LIN {X 0,Y 480.897,Z 537.281,A -85,B 0,C 180,E1 -6841.675,E2 -6841.675} C_VEL
LIN {X 0,Y 481.01,Z 535.652,A -85,B 0,C 180,E1 -6843.35,E2 -6843.35} C_VEL
LIN {X 0,Y 481.08,Z 532.877,A -85,B 0,C 180,E1 -6845.029,E2 -6845.029} C_VEL
LIN {X 0,Y 481.293,Z 528.594,A -85,B 0,C 180,E1 -6846.803,E2 -6846.803} C_VEL
LIN {X 0,Y 481.489,Z 523.502,A -85,B 0,C 180,E1 -6848.393,E2 -6848.393} C_VEL
LIN {X 0,Y 481.749,Z 516.626,A -85,B 0,C 180,E1 -6850.082,E2 -6850.082} C_VEL
LIN {X 0,Y 482.2,Z 509.189,A -85,B 0,C 180,E1 -6851.561,E2 -6851.561} C_VEL
LIN {X 0,Y 482.622,Z 500.167,A -85,B 0,C 180,E1 -6853.045,E2 -6853.045} C_VEL
LIN {X 0,Y 483.158,Z 490.915,A -85,B 0,C 180,E1 -6854.317,E2 -6854.317} C_VEL
LIN {X 0,Y 483.742,Z 479.844,A -85,B 0,C 180,E1 -6855.591,E2 -6855.591} C_VEL
LIN {X 0,Y 484.392,Z 467.732,A -85,B 0,C 180,E1 -6856.746,E2 -6856.746} C_VEL
LIN {X 0,Y 484.961,Z 455.431,A -85,B 0,C 180,E1 -6857.718,E2 -6857.718} C_VEL
LIN {X 0,Y 485.59,Z 440.986,A -85,B 0,C 180,E1 -6858.638,E2 -6858.638} C_VEL
LIN {X 0,Y 485.834,Z 427.276,A -85,B 0,C 180,E1 -6859.339,E2 -6859.339} C_VEL
LIN {X 0,Y 481.687,Z 414.112,A -85,B 0,C 180,E1 -6860.052,E2 -6860.052} C_VEL
LIN {X 0,Y 481.666,Z 414.111,A -85,B 0,C 180,E1 -6863.201,E2 -6863.201} C_VEL
LIN {X 0,Y 481.691,Z 414.114,A -85,B 0,C 180,E1 -6865.958,E2 -6865.958} C_VEL
LIN {X 0,Y 481.702,Z 414.107,A -85,B 0,C 180,E1 -6868.781,E2 -6868.781} C_VEL
LIN {X 0,Y 481.661,Z 414.113,A -85,B 0,C 180,E1 -6872.19,E2 -6872.19} C_VEL
LIN {X 0,Y 481.69,Z 414.107,A -85,B 0,C 180,E1 -6874.682,E2 -6874.682} C_VEL
LIN {X 0,Y 481.656,Z 414.115,A -85,B 0,C 180,E1 -6878.007,E2 -6878.007} C_VEL
LIN {X 0,Y 481.664,Z 414.113,A -85,B 0,C 180,E1 -6881.041,E2 -6881.041} C_VEL
LIN {X 0,Y 481.738,Z 414.259,A -85,B 0,C 180,E1 -6884.055,E2 -6884.055} C_VEL
LIN {X 0,Y 481.86,Z 418.445,A -85,B 0,C 180,E1 -6885.616,E2 -6885.616} C_VEL
LIN {X 0,Y 481.614,Z 430.552,A -85,B 0,C 180,E1 -6889.71,E2 -6889.71} C_VEL
LIN {X 0,Y 481.795,Z 440.07,A -85,B 0,C 180,E1 -6892.745,E2 -6892.745} C_VEL
LIN {X 0,Y 481.916,Z 449.965,A -85,B 0,C 180,E1 -6895.817,E2 -6895.817} C_VEL
LIN {X 0,Y 481.956,Z 459.783,A -85,B 0,C 180,E1 -6898.824,E2 -6898.824} C_VEL
LIN {X 0,Y 481.976,Z 469.257,A -85,B 0,C 180,E1 -6901.712,E2 -6901.712} C_VEL
LIN {X 0,Y 481.793,Z 479.207,A -85,B 0,C 180,E1 -6904.743,E2 -6904.743} C_VEL
LIN {X 0,Y 481.638,Z 488.806,A -85,B 0,C 180,E1 -6907.704,E2 -6907.704} C_VEL
LIN {X 0,Y 481.504,Z 497.467,A -85,B 0,C 180,E1 -6910.384,E2 -6910.384} C_VEL
LIN {X 0,Y 481.447,Z 502.384,A -85,B 0,C 180,E1 -6911.923,E2 -6911.923} C_VEL
LIN {X 0,Y 484.792,Z 518.216,A -85,B 0,C 180,E1 -6912.407,E2 -6912.407} C_VEL
LIN {X 0,Y 485.454,Z 522.705,A -85,B 0,C 180,E1 -6912.57,E2 -6912.57} C_VEL
LIN {X 0,Y 485.075,Z 535.599,A -85,B 0,C 180,E1 -6913.058,E2 -6913.058} C_VEL
LIN {X 0,Y 484.495,Z 549.866,A -85,B 0,C 180,E1 -6913.785,E2 -6913.785} C_VEL
LIN {X 0,Y 483.935,Z 562.713,A -85,B 0,C 180,E1 -6914.631,E2 -6914.631} C_VEL
LIN {X 0,Y 483.286,Z 574.358,A -85,B 0,C 180,E1 -6915.58,E2 -6915.58} C_VEL
LIN {X 0,Y 482.67,Z 585.939,A -85,B 0,C 180,E1 -6916.742,E2 -6916.742} C_VEL
LIN {X 0,Y 482.228,Z 596.661,A -85,B 0,C 180,E1 -6918.062,E2 -6918.062} C_VEL
LIN {X 0,Y 481.671,Z 606.186,A -85,B 0,C 180,E1 -6919.491,E2 -6919.491} C_VEL
LIN {X 0,Y 481.328,Z 614.151,A -85,B 0,C 180,E1 -6920.969,E2 -6920.969} C_VEL
LIN {X 0,Y 481.054,Z 620.547,A -85,B 0,C 180,E1 -6922.445,E2 -6922.445} C_VEL
LIN {X 0,Y 480.951,Z 626.202,A -85,B 0,C 180,E1 -6924.129,E2 -6924.129} C_VEL
LIN {X 0,Y 480.817,Z 630.31,A -85,B 0,C 180,E1 -6925.809,E2 -6925.809} C_VEL
LIN {X 0,Y 480.879,Z 631.825,A -85,B 0,C 180,E1 -6926.649,E2 -6926.649} C_VEL
LIN {X 0,Y 480.786,Z 633.83,A -85,B 0,C 180,E1 -6928.325,E2 -6928.325} C_VEL
LIN {X 0,Y 480.741,Z 634.5,A -85,B 0,C 180,E1 -6930,E2 -6930} C_VEL
LIN {X 0,Y 480.786,Z 633.827,A -85,B 0,C 180,E1 -6931.675,E2 -6931.675} C_VEL
LIN {X 0,Y 480.879,Z 631.826,A -85,B 0,C 180,E1 -6933.351,E2 -6933.351} C_VEL
LIN {X 0,Y 480.896,Z 628.445,A -85,B 0,C 180,E1 -6935.031,E2 -6935.031} C_VEL
LIN {X 0,Y 480.996,Z 623.596,A -85,B 0,C 180,E1 -6936.713,E2 -6936.713} C_VEL
LIN {X 0,Y 481.141,Z 618.859,A -85,B 0,C 180,E1 -6937.976,E2 -6937.976} C_VEL
LIN {X 0,Y 481.426,Z 612.055,A -85,B 0,C 180,E1 -6939.453,E2 -6939.453} C_VEL
LIN {X 0,Y 481.833,Z 603.569,A -85,B 0,C 180,E1 -6940.93,E2 -6940.93} C_VEL
LIN {X 0,Y 482.258,Z 593.829,A -85,B 0,C 180,E1 -6942.315,E2 -6942.315} C_VEL
LIN {X 0,Y 482.793,Z 583.991,A -85,B 0,C 180,E1 -6943.469,E2 -6943.469} C_VEL
LIN {X 0,Y 483.314,Z 573.157,A -85,B 0,C 180,E1 -6944.527,E2 -6944.527} C_VEL
LIN {X 0,Y 483.986,Z 561.269,A -85,B 0,C 180,E1 -6945.475,E2 -6945.475} C_VEL
LIN {X 0,Y 484.586,Z 548.033,A -85,B 0,C 180,E1 -6946.32,E2 -6946.32} C_VEL
LIN {X 0,Y 485.074,Z 535.108,A -85,B 0,C 180,E1 -6946.963,E2 -6946.963} C_VEL
LIN {X 0,Y 485.341,Z 521.153,A -85,B 0,C 180,E1 -6947.486,E2 -6947.486} C_VEL
LIN {X 0,Y 482.502,Z 507.123,A -85,B 0,C 180,E1 -6947.951,E2 -6947.951} C_VEL
LIN {X 0,Y 481.446,Z 502.32,A -85,B 0,C 180,E1 -6948.096,E2 -6948.096} C_VEL
LIN {X 0,Y 481.641,Z 492.574,A -85,B 0,C 180,E1 -6951.395,E2 -6951.395} C_VEL
LIN {X 0,Y 481.85,Z 483.299,A -85,B 0,C 180,E1 -6954.563,E2 -6954.563} C_VEL
LIN {X 0,Y 482.004,Z 475.751,A -85,B 0,C 180,E1 -6957.198,E2 -6957.198} C_VEL
LIN {X 0,Y 482.218,Z 468.781,A -85,B 0,C 180,E1 -6959.705,E2 -6959.705} C_VEL
LIN {X 0,Y 482.438,Z 460.823,A -85,B 0,C 180,E1 -6962.616,E2 -6962.616} C_VEL
LIN {X 0,Y 482.647,Z 452.865,A -85,B 0,C 180,E1 -6965.623,E2 -6965.623} C_VEL
LIN {X 0,Y 482.809,Z 444.905,A -85,B 0,C 180,E1 -6968.75,E2 -6968.75} C_VEL
LIN {X 0,Y 483.014,Z 438.229,A -85,B 0,C 180,E1 -6971.456,E2 -6971.456} C_VEL
LIN {X 0,Y 483.396,Z 429.907,A -85,B 0,C 180,E1 -6974.947,E2 -6974.947} C_VEL
LIN {X 0,Y 483.455,Z 425.426,A -85,B 0,C 180,E1 -6976.903,E2 -6976.903} C_VEL
LIN {X 0,Y 482.819,Z 420.482,A -85,B 0,C 180,E1 -6979.194,E2 -6979.194} C_VEL
LIN {X 0,Y 481.671,Z 414.114,A -85,B 0,C 180,E1 -6982.339,E2 -6982.339} C_VEL
LIN {X 0,Y 481.694,Z 414.11,A -85,B 0,C 180,E1 -6985.318,E2 -6985.318} C_VEL
LIN {X 0,Y 481.647,Z 414.118,A -85,B 0,C 180,E1 -6988.312,E2 -6988.312} C_VEL
LIN {X 0,Y 481.702,Z 414.111,A -85,B 0,C 180,E1 -6991.219,E2 -6991.219} C_VEL
LIN {X 0,Y 481.703,Z 414.101,A -85,B 0,C 180,E1 -6994.043,E2 -6994.043} C_VEL
LIN {X 0,Y 481.676,Z 414.11,A -85,B 0,C 180,E1 -6996.812,E2 -6996.812} C_VEL
LIN {X 0,Y 481.699,Z 414.1,A -85,B 0,C 180,E1 -6999.503,E2 -6999.503} C_VEL
LIN {X 0,Y 481.71,Z 414.108,A -85,B 0,C 180,E1 -7002.159,E2 -7002.159} C_VEL
LIN {X 0,Y 481.745,Z 414.097,A -85,B 0,C 180,E1 -7004.776,E2 -7004.776} C_VEL
LIN {X 0,Y 481.753,Z 414.102,A -85,B 0,C 180,E1 -7008.215,E2 -7008.215} C_VEL
LIN {X 0,Y 481.743,Z 414.095,A -85,B 0,C 180,E1 -7011.611,E2 -7011.611} C_VEL
LIN {X 0,Y 481.819,Z 414.095,A -85,B 0,C 180,E1 -7014.14,E2 -7014.14} C_VEL
LIN {X 0,Y 481.93,Z 414.073,A -85,B 0,C 180,E1 -7017.493,E2 -7017.493} C_VEL
LIN {X 0,Y 481.908,Z 414.081,A -85,B 0,C 180,E1 -7020.836,E2 -7020.836} C_VEL
LIN {X 0,Y 481.929,Z 414.074,A -85,B 0,C 180,E1 -7022.508,E2 -7022.508} C_VEL
LIN {X 0,Y 481.818,Z 414.095,A -85,B 0,C 180,E1 -7025.86,E2 -7025.86} C_VEL
LIN {X 0,Y 481.765,Z 414.092,A -85,B 0,C 180,E1 -7028.388,E2 -7028.388} C_VEL
LIN {X 0,Y 481.753,Z 414.103,A -85,B 0,C 180,E1 -7031.785,E2 -7031.785} C_VEL
LIN {X 0,Y 481.745,Z 414.104,A -85,B 0,C 180,E1 -7035.224,E2 -7035.224} C_VEL
LIN {X 0,Y 481.715,Z 414.1,A -85,B 0,C 180,E1 -7038.722,E2 -7038.722} C_VEL
LIN {X 0,Y 481.648,Z 414.114,A -85,B 0,C 180,E1 -7041.395,E2 -7041.395} C_VEL
LIN {X 0,Y 481.663,Z 414.114,A -85,B 0,C 180,E1 -7044.114,E2 -7044.114} C_VEL
LIN {X 0,Y 481.749,Z 414.101,A -85,B 0,C 180,E1 -7047.139,E2 -7047.139} C_VEL
LIN {X 0,Y 481.681,Z 414.11,A -85,B 0,C 180,E1 -7049.741,E2 -7049.741} C_VEL
LIN {X 0,Y 481.674,Z 414.111,A -85,B 0,C 180,E1 -7052.674,E2 -7052.674} C_VEL
LIN {X 0,Y 481.638,Z 414.114,A -85,B 0,C 180,E1 -7055.71,E2 -7055.71} C_VEL
LIN {X 0,Y 481.673,Z 414.113,A -85,B 0,C 180,E1 -7058.859,E2 -7058.859} C_VEL
LIN {X 0,Y 481.664,Z 414.114,A -85,B 0,C 180,E1 -7061.914,E2 -7061.914} C_VEL
LIN {X 0,Y 481.662,Z 414.112,A -85,B 0,C 180,E1 -7064.457,E2 -7064.457} C_VEL
LIN {X 0,Y 481.65,Z 414.12,A -85,B 0,C 180,E1 -7067.839,E2 -7067.839} C_VEL
LIN {X 0,Y 481.751,Z 414.254,A -85,B 0,C 180,E1 -7069.263,E2 -7069.263} C_VEL
LIN {X 0,Y 482.904,Z 420.934,A -85,B 0,C 180,E1 -7071.259,E2 -7071.259} C_VEL
LIN {X 0,Y 482.976,Z 427.428,A -85,B 0,C 180,E1 -7073.162,E2 -7073.162} C_VEL
LIN {X 0,Y 482.647,Z 438.338,A -85,B 0,C 180,E1 -7076.404,E2 -7076.404} C_VEL
LIN {X 0,Y 482.528,Z 448.105,A -85,B 0,C 180,E1 -7079.351,E2 -7079.351} C_VEL
LIN {X 0,Y 482.356,Z 457.601,A -85,B 0,C 180,E1 -7082.209,E2 -7082.209} C_VEL
LIN {X 0,Y 482.025,Z 468.434,A -85,B 0,C 180,E1 -7085.427,E2 -7085.427} C_VEL
LIN {X 0,Y 481.305,Z 470.724,A -85,B 0,C 180,E1 -7086.069,E2 -7086.069} C_VEL
LIN {X 0,Y 475.485,Z 478.674,A -85,B 0,C 180,E1 -7088.137,E2 -7088.137} C_VEL
LIN {X 0,Y 474.804,Z 481.025,A -85,B 0,C 180,E1 -7088.789,E2 -7088.789} C_VEL
LIN {X 0,Y 474.606,Z 491.302,A -85,B 0,C 180,E1 -7091.683,E2 -7091.683} C_VEL
LIN {X 0,Y 478.17,Z 508.468,A -85,B 0,C 180,E1 -7092.207,E2 -7092.207} C_VEL
LIN {X 0,Y 478.686,Z 513.051,A -85,B 0,C 180,E1 -7092.374,E2 -7092.374} C_VEL
LIN {X 0,Y 478.21,Z 526.916,A -85,B 0,C 180,E1 -7092.907,E2 -7092.907} C_VEL
LIN {X 0,Y 477.764,Z 539.465,A -85,B 0,C 180,E1 -7093.556,E2 -7093.556} C_VEL
LIN {X 0,Y 477.121,Z 552.398,A -85,B 0,C 180,E1 -7094.406,E2 -7094.406} C_VEL
LIN {X 0,Y 476.544,Z 562.958,A -85,B 0,C 180,E1 -7095.262,E2 -7095.262} C_VEL
LIN {X 0,Y 475.905,Z 573.916,A -85,B 0,C 180,E1 -7096.333,E2 -7096.333} C_VEL
LIN {X 0,Y 475.285,Z 584.287,A -85,B 0,C 180,E1 -7097.564,E2 -7097.564} C_VEL
LIN {X 0,Y 474.865,Z 593.594,A -85,B 0,C 180,E1 -7098.907,E2 -7098.907} C_VEL
LIN {X 0,Y 474.416,Z 602.109,A -85,B 0,C 180,E1 -7100.406,E2 -7100.406} C_VEL
LIN {X 0,Y 474.084,Z 608.977,A -85,B 0,C 180,E1 -7101.904,E2 -7101.904} C_VEL
LIN {X 0,Y 473.923,Z 614.762,A -85,B 0,C 180,E1 -7103.501,E2 -7103.501} C_VEL
LIN {X 0,Y 473.837,Z 618.639,A -85,B 0,C 180,E1 -7104.894,E2 -7104.894} C_VEL
LIN {X 0,Y 473.788,Z 622.059,A -85,B 0,C 180,E1 -7106.598,E2 -7106.598} C_VEL
LIN {X 0,Y 473.694,Z 624.095,A -85,B 0,C 180,E1 -7108.3,E2 -7108.3} C_VEL
LIN {X 0,Y 473.668,Z 624.799,A -85,B 0,C 180,E1 -7110,E2 -7110} C_VEL
LIN {X 0,Y 473.692,Z 624.175,A -85,B 0,C 180,E1 -7111.7,E2 -7111.7} C_VEL
LIN {X 0,Y 473.788,Z 622.207,A -85,B 0,C 180,E1 -7113.402,E2 -7113.402} C_VEL
LIN {X 0,Y 473.836,Z 618.858,A -85,B 0,C 180,E1 -7115.106,E2 -7115.106} C_VEL
LIN {X 0,Y 473.925,Z 614.029,A -85,B 0,C 180,E1 -7116.813,E2 -7116.813} C_VEL
LIN {X 0,Y 474.16,Z 607.57,A -85,B 0,C 180,E1 -7118.524,E2 -7118.524} C_VEL
LIN {X 0,Y 474.472,Z 600.372,A -85,B 0,C 180,E1 -7120.023,E2 -7120.023} C_VEL
LIN {X 0,Y 475.003,Z 591.412,A -85,B 0,C 180,E1 -7121.522,E2 -7121.522} C_VEL
LIN {X 0,Y 475.466,Z 582.037,A -85,B 0,C 180,E1 -7122.81,E2 -7122.81} C_VEL
LIN {X 0,Y 476.056,Z 571.663,A -85,B 0,C 180,E1 -7123.99,E2 -7123.99} C_VEL
LIN {X 0,Y 476.658,Z 560.22,A -85,B 0,C 180,E1 -7125.062,E2 -7125.062} C_VEL
LIN {X 0,Y 477.346,Z 547.551,A -85,B 0,C 180,E1 -7126.025,E2 -7126.025} C_VEL
LIN {X 0,Y 477.887,Z 535.604,A -85,B 0,C 180,E1 -7126.751,E2 -7126.751} C_VEL
LIN {X 0,Y 478.384,Z 521.502,A -85,B 0,C 180,E1 -7127.417,E2 -7127.417} C_VEL
LIN {X 0,Y 478.613,Z 510.719,A -85,B 0,C 180,E1 -7127.795,E2 -7127.795} C_VEL
LIN {X 0,Y 475.665,Z 496.343,A -85,B 0,C 180,E1 -7128.268,E2 -7128.268} C_VEL
LIN {X 0,Y 474.627,Z 491.285,A -85,B 0,C 180,E1 -7128.41,E2 -7128.41} C_VEL
LIN {X 0,Y 474.831,Z 479.581,A -85,B 0,C 180,E1 -7131.717,E2 -7131.717} C_VEL
LIN {X 0,Y 475.031,Z 468.587,A -85,B 0,C 180,E1 -7134.939,E2 -7134.939} C_VEL
LIN {X 0,Y 475.308,Z 459.023,A -85,B 0,C 180,E1 -7137.807,E2 -7137.807} C_VEL
LIN {X 0,Y 475.517,Z 448.532,A -85,B 0,C 180,E1 -7140.994,E2 -7140.994} C_VEL
LIN {X 0,Y 475.673,Z 439.835,A -85,B 0,C 180,E1 -7143.646,E2 -7143.646} C_VEL
LIN {X 0,Y 476.061,Z 427.824,A -85,B 0,C 180,E1 -7147.249,E2 -7147.249} C_VEL
LIN {X 0,Y 475.908,Z 422.197,A -85,B 0,C 180,E1 -7148.923,E2 -7148.923} C_VEL
LIN {X 0,Y 474.64,Z 414.992,A -85,B 0,C 180,E1 -7151.118,E2 -7151.118} C_VEL
LIN {X 0,Y 474.612,Z 414.992,A -85,B 0,C 180,E1 -7154.105,E2 -7154.105} C_VEL
LIN {X 0,Y 474.643,Z 414.993,A -85,B 0,C 180,E1 -7157.069,E2 -7157.069} C_VEL
LIN {X 0,Y 474.646,Z 414.989,A -85,B 0,C 180,E1 -7160.454,E2 -7160.454} C_VEL
LIN {X 0,Y 474.595,Z 414.993,A -85,B 0,C 180,E1 -7163.677,E2 -7163.677} C_VEL
LIN {X 0,Y 474.645,Z 414.987,A -85,B 0,C 180,E1 -7166.78,E2 -7166.78} C_VEL
LIN {X 0,Y 474.615,Z 414.984,A -85,B 0,C 180,E1 -7169.77,E2 -7169.77} C_VEL
LIN {X 0,Y 474.699,Z 414.983,A -85,B 0,C 180,E1 -7172.68,E2 -7172.68} C_VEL
LIN {X 0,Y 474.662,Z 414.984,A -85,B 0,C 180,E1 -7175.507,E2 -7175.507} C_VEL
LIN {X 0,Y 474.673,Z 414.985,A -85,B 0,C 180,E1 -7179.185,E2 -7179.185} C_VEL
LIN {X 0,Y 474.649,Z 414.994,A -85,B 0,C 180,E1 -7179.694,E2 -7179.694} C_VEL
LIN {X 0,Y 479.11,Z 428.79,A -85,B 0,C 180,E1 -7180.487,E2 -7180.487} C_VEL
LIN {X 0,Y 479.317,Z 431.283,A -85,B 0,C 180,E1 -7180.621,E2 -7180.621} C_VEL
LIN {X 0,Y 478.741,Z 444.726,A -85,B 0,C 180,E1 -7181.38,E2 -7181.38} C_VEL
LIN {X 0,Y 478.025,Z 458.574,A -85,B 0,C 180,E1 -7182.348,E2 -7182.348} C_VEL
LIN {X 0,Y 477.353,Z 470.767,A -85,B 0,C 180,E1 -7183.389,E2 -7183.389} C_VEL
LIN {X 0,Y 476.645,Z 482.694,A -85,B 0,C 180,E1 -7184.609,E2 -7184.609} C_VEL
LIN {X 0,Y 476.047,Z 493.244,A -85,B 0,C 180,E1 -7185.901,E2 -7185.901} C_VEL
LIN {X 0,Y 475.397,Z 503.14,A -85,B 0,C 180,E1 -7187.345,E2 -7187.345} C_VEL
LIN {X 0,Y 474.944,Z 512.005,A -85,B 0,C 180,E1 -7188.909,E2 -7188.909} C_VEL
LIN {X 0,Y 474.541,Z 519.939,A -85,B 0,C 180,E1 -7190.624,E2 -7190.624} C_VEL
LIN {X 0,Y 474.275,Z 526.241,A -85,B 0,C 180,E1 -7192.336,E2 -7192.336} C_VEL
LIN {X 0,Y 474.086,Z 531.121,A -85,B 0,C 180,E1 -7194.044,E2 -7194.044} C_VEL
LIN {X 0,Y 474.06,Z 534.702,A -85,B 0,C 180,E1 -7195.749,E2 -7195.749} C_VEL
LIN {X 0,Y 473.903,Z 537.101,A -85,B 0,C 180,E1 -7197.45,E2 -7197.45} C_VEL
LIN {X 0,Y 473.782,Z 538.359,A -85,B 0,C 180,E1 -7199.15,E2 -7199.15} C_VEL
LIN {X 0,Y 473.786,Z 538.445,A -85,B 0,C 180,E1 -7200.85,E2 -7200.85} C_VEL
LIN {X 0,Y 473.916,Z 537.378,A -85,B 0,C 180,E1 -7202.55,E2 -7202.55} C_VEL
LIN {X 0,Y 474.08,Z 535.175,A -85,B 0,C 180,E1 -7204.251,E2 -7204.251} C_VEL
LIN {X 0,Y 474.193,Z 531.789,A -85,B 0,C 180,E1 -7205.955,E2 -7205.955} C_VEL
LIN {X 0,Y 474.335,Z 527.111,A -85,B 0,C 180,E1 -7207.663,E2 -7207.663} C_VEL
LIN {X 0,Y 474.603,Z 520.989,A -85,B 0,C 180,E1 -7209.375,E2 -7209.375} C_VEL
LIN {X 0,Y 475.027,Z 513.236,A -85,B 0,C 180,E1 -7211.089,E2 -7211.089} C_VEL
LIN {X 0,Y 475.419,Z 505.604,A -85,B 0,C 180,E1 -7212.479,E2 -7212.479} C_VEL
LIN {X 0,Y 475.988,Z 496.355,A -85,B 0,C 180,E1 -7213.883,E2 -7213.883} C_VEL
LIN {X 0,Y 476.565,Z 486.188,A -85,B 0,C 180,E1 -7215.175,E2 -7215.175} C_VEL
LIN {X 0,Y 477.189,Z 474.818,A -85,B 0,C 180,E1 -7216.381,E2 -7216.381} C_VEL
LIN {X 0,Y 477.945,Z 462.818,A -85,B 0,C 180,E1 -7217.434,E2 -7217.434} C_VEL
LIN {X 0,Y 478.507,Z 449.439,A -85,B 0,C 180,E1 -7218.408,E2 -7218.408} C_VEL
LIN {X 0,Y 479.076,Z 435.711,A -85,B 0,C 180,E1 -7219.208,E2 -7219.208} C_VEL
LIN {X 0,Y 479.206,Z 429.405,A -85,B 0,C 180,E1 -7219.521,E2 -7219.521} C_VEL
LIN {X 0,Y 474.66,Z 414.987,A -85,B 0,C 180,E1 -7220.334,E2 -7220.334} C_VEL
LIN {X 0,Y 474.611,Z 414.992,A -85,B 0,C 180,E1 -7223.566,E2 -7223.566} C_VEL
LIN {X 0,Y 474.656,Z 414.987,A -85,B 0,C 180,E1 -7226.372,E2 -7226.372} C_VEL
LIN {X 0,Y 474.623,Z 414.99,A -85,B 0,C 180,E1 -7229.252,E2 -7229.252} C_VEL
LIN {X 0,Y 474.619,Z 414.989,A -85,B 0,C 180,E1 -7232.431,E2 -7232.431} C_VEL
LIN {X 0,Y 474.616,Z 414.993,A -85,B 0,C 180,E1 -7235.469,E2 -7235.469} C_VEL
LIN {X 0,Y 474.613,Z 414.989,A -85,B 0,C 180,E1 -7238.457,E2 -7238.457} C_VEL
LIN {X 0,Y 474.634,Z 414.988,A -85,B 0,C 180,E1 -7240.96,E2 -7240.96} C_VEL
LIN {X 0,Y 474.669,Z 415.047,A -85,B 0,C 180,E1 -7243.841,E2 -7243.841} C_VEL
LIN {X 0,Y 474.922,Z 418.667,A -85,B 0,C 180,E1 -7245.261,E2 -7245.261} C_VEL
LIN {X 0,Y 474.549,Z 430.316,A -85,B 0,C 180,E1 -7249.335,E2 -7249.335} C_VEL
LIN {X 0,Y 474.737,Z 440.38,A -85,B 0,C 180,E1 -7252.63,E2 -7252.63} C_VEL
LIN {X 0,Y 474.848,Z 450.312,A -85,B 0,C 180,E1 -7255.777,E2 -7255.777} C_VEL
LIN {X 0,Y 474.871,Z 460.011,A -85,B 0,C 180,E1 -7258.802,E2 -7258.802} C_VEL
LIN {X 0,Y 474.871,Z 469.463,A -85,B 0,C 180,E1 -7261.732,E2 -7261.732} C_VEL
LIN {X 0,Y 474.726,Z 478.656,A -85,B 0,C 180,E1 -7264.575,E2 -7264.575} C_VEL
LIN {X 0,Y 474.585,Z 487.536,A -85,B 0,C 180,E1 -7267.355,E2 -7267.355} C_VEL
LIN {X 0,Y 474.448,Z 496.22,A -85,B 0,C 180,E1 -7270.081,E2 -7270.081} C_VEL
LIN {X 0,Y 474.373,Z 501.021,A -85,B 0,C 180,E1 -7271.593,E2 -7271.593} C_VEL
LIN {X 0,Y 474.956,Z 504.896,A -85,B 0,C 180,E1 -7271.706,E2 -7271.706} C_VEL
LIN {X 0,Y 478.23,Z 520.495,A -85,B 0,C 180,E1 -7272.235,E2 -7272.235} C_VEL
LIN {X 0,Y 478.639,Z 524.063,A -85,B 0,C 180,E1 -7272.372,E2 -7272.372} C_VEL
LIN {X 0,Y 478.201,Z 537.422,A -85,B 0,C 180,E1 -7272.906,E2 -7272.906} C_VEL
LIN {X 0,Y 477.583,Z 551.63,A -85,B 0,C 180,E1 -7273.658,E2 -7273.658} C_VEL
LIN {X 0,Y 477.008,Z 564.126,A -85,B 0,C 180,E1 -7274.512,E2 -7274.512} C_VEL
LIN {X 0,Y 476.314,Z 575.491,A -85,B 0,C 180,E1 -7275.473,E2 -7275.473} C_VEL
LIN {X 0,Y 475.731,Z 585.936,A -85,B 0,C 180,E1 -7276.545,E2 -7276.545} C_VEL
LIN {X 0,Y 475.235,Z 596.076,A -85,B 0,C 180,E1 -7277.803,E2 -7277.803} C_VEL
LIN {X 0,Y 474.74,Z 604.878,A -85,B 0,C 180,E1 -7279.12,E2 -7279.12} C_VEL
LIN {X 0,Y 474.327,Z 613.099,A -85,B 0,C 180,E1 -7280.62,E2 -7280.62} C_VEL
LIN {X 0,Y 474.079,Z 618.844,A -85,B 0,C 180,E1 -7281.904,E2 -7281.904} C_VEL
LIN {X 0,Y 473.877,Z 624.749,A -85,B 0,C 180,E1 -7283.549,E2 -7283.549} C_VEL
LIN {X 0,Y 473.831,Z 628.44,A -85,B 0,C 180,E1 -7284.894,E2 -7284.894} C_VEL
LIN {X 0,Y 473.787,Z 631.825,A -85,B 0,C 180,E1 -7286.598,E2 -7286.598} C_VEL
LIN {X 0,Y 473.692,Z 633.83,A -85,B 0,C 180,E1 -7288.3,E2 -7288.3} C_VEL
LIN {X 0,Y 473.668,Z 634.5,A -85,B 0,C 180,E1 -7290,E2 -7290} C_VEL
LIN {X 0,Y 473.692,Z 633.827,A -85,B 0,C 180,E1 -7291.7,E2 -7291.7} C_VEL
LIN {X 0,Y 473.787,Z 631.825,A -85,B 0,C 180,E1 -7293.402,E2 -7293.402} C_VEL
LIN {X 0,Y 473.83,Z 628.444,A -85,B 0,C 180,E1 -7295.106,E2 -7295.106} C_VEL
LIN {X 0,Y 473.908,Z 623.598,A -85,B 0,C 180,E1 -7296.814,E2 -7296.814} C_VEL
LIN {X 0,Y 474.08,Z 618.858,A -85,B 0,C 180,E1 -7298.096,E2 -7298.096} C_VEL
LIN {X 0,Y 474.399,Z 612.055,A -85,B 0,C 180,E1 -7299.594,E2 -7299.594} C_VEL
LIN {X 0,Y 474.826,Z 603.568,A -85,B 0,C 180,E1 -7301.094,E2 -7301.094} C_VEL
LIN {X 0,Y 475.244,Z 594.472,A -85,B 0,C 180,E1 -7302.414,E2 -7302.414} C_VEL
LIN {X 0,Y 475.866,Z 583.991,A -85,B 0,C 180,E1 -7303.668,E2 -7303.668} C_VEL
LIN {X 0,Y 476.413,Z 573.157,A -85,B 0,C 180,E1 -7304.742,E2 -7304.742} C_VEL
LIN {X 0,Y 477.144,Z 561.249,A -85,B 0,C 180,E1 -7305.703,E2 -7305.703} C_VEL
LIN {X 0,Y 477.729,Z 548.153,A -85,B 0,C 180,E1 -7306.547,E2 -7306.547} C_VEL
LIN {X 0,Y 478.293,Z 534.458,A -85,B 0,C 180,E1 -7307.233,E2 -7307.233} C_VEL
LIN {X 0,Y 478.5,Z 521.835,A -85,B 0,C 180,E1 -7307.716,E2 -7307.716} C_VEL
LIN {X 0,Y 475.433,Z 506.779,A -85,B 0,C 180,E1 -7308.243,E2 -7308.243} C_VEL
LIN {X 0,Y 474.349,Z 501.792,A -85,B 0,C 180,E1 -7308.38,E2 -7308.38} C_VEL
LIN {X 0,Y 474.593,Z 492.048,A -85,B 0,C 180,E1 -7311.729,E2 -7311.729} C_VEL
LIN {X 0,Y 474.809,Z 482.761,A -85,B 0,C 180,E1 -7314.951,E2 -7314.951} C_VEL
LIN {X 0,Y 475.051,Z 473.554,A -85,B 0,C 180,E1 -7318.256,E2 -7318.256} C_VEL
LIN {X 0,Y 475.272,Z 465.632,A -85,B 0,C 180,E1 -7321.169,E2 -7321.169} C_VEL
LIN {X 0,Y 475.491,Z 457.689,A -85,B 0,C 180,E1 -7324.171,E2 -7324.171} C_VEL
LIN {X 0,Y 475.689,Z 450.253,A -85,B 0,C 180,E1 -7327.078,E2 -7327.078} C_VEL
LIN {X 0,Y 475.977,Z 441.747,A -85,B 0,C 180,E1 -7330.517,E2 -7330.517} C_VEL
LIN {X 0,Y 476.271,Z 433.674,A -85,B 0,C 180,E1 -7333.912,E2 -7333.912} C_VEL
LIN {X 0,Y 476.526,Z 428.23,A -85,B 0,C 180,E1 -7336.276,E2 -7336.276} C_VEL
LIN {X 0,Y 476.156,Z 423.643,A -85,B 0,C 180,E1 -7338.379,E2 -7338.379} C_VEL
LIN {X 0,Y 474.986,Z 416.935,A -85,B 0,C 180,E1 -7341.647,E2 -7341.647} C_VEL
LIN {X 0,Y 474.618,Z 414.991,A -85,B 0,C 180,E1 -7342.688,E2 -7342.688} C_VEL
LIN {X 0,Y 474.64,Z 414.987,A -85,B 0,C 180,E1 -7346.016,E2 -7346.016} C_VEL
LIN {X 0,Y 474.606,Z 414.992,A -85,B 0,C 180,E1 -7349.19,E2 -7349.19} C_VEL
LIN {X 0,Y 474.699,Z 414.981,A -85,B 0,C 180,E1 -7352.68,E2 -7352.68} C_VEL
LIN {X 0,Y 474.661,Z 414.982,A -85,B 0,C 180,E1 -7355.507,E2 -7355.507} C_VEL
LIN {X 0,Y 474.673,Z 414.976,A -85,B 0,C 180,E1 -7359.186,E2 -7359.186} C_VEL
LIN {X 0,Y 474.659,Z 414.987,A -85,B 0,C 180,E1 -7361.884,E2 -7361.884} C_VEL
LIN {X 0,Y 474.702,Z 414.975,A -85,B 0,C 180,E1 -7364.544,E2 -7364.544} C_VEL
LIN {X 0,Y 474.707,Z 414.982,A -85,B 0,C 180,E1 -7368.038,E2 -7368.038} C_VEL
LIN {X 0,Y 474.714,Z 414.971,A -85,B 0,C 180,E1 -7371.486,E2 -7371.486} C_VEL
LIN {X 0,Y 474.781,Z 414.972,A -85,B 0,C 180,E1 -7374.052,E2 -7374.052} C_VEL
LIN {X 0,Y 474.896,Z 414.949,A -85,B 0,C 180,E1 -7377.455,E2 -7377.455} C_VEL
LIN {X 0,Y 474.914,Z 414.956,A -85,B 0,C 180,E1 -7380,E2 -7380} C_VEL
LIN {X 0,Y 474.895,Z 414.95,A -85,B 0,C 180,E1 -7382.545,E2 -7382.545} C_VEL
LIN {X 0,Y 474.781,Z 414.973,A -85,B 0,C 180,E1 -7385.948,E2 -7385.948} C_VEL
LIN {X 0,Y 474.731,Z 414.968,A -85,B 0,C 180,E1 -7388.514,E2 -7388.514} C_VEL
LIN {X 0,Y 474.707,Z 414.982,A -85,B 0,C 180,E1 -7391.962,E2 -7391.962} C_VEL
LIN {X 0,Y 474.702,Z 414.98,A -85,B 0,C 180,E1 -7395.456,E2 -7395.456} C_VEL
LIN {X 0,Y 474.668,Z 414.978,A -85,B 0,C 180,E1 -7399.01,E2 -7399.01} C_VEL
LIN {X 0,Y 474.59,Z 414.992,A -85,B 0,C 180,E1 -7401.729,E2 -7401.729} C_VEL
LIN {X 0,Y 474.643,Z 414.987,A -85,B 0,C 180,E1 -7404.494,E2 -7404.494} C_VEL
LIN {X 0,Y 474.701,Z 414.98,A -85,B 0,C 180,E1 -7407.339,E2 -7407.339} C_VEL
LIN {X 0,Y 474.606,Z 414.99,A -85,B 0,C 180,E1 -7410.81,E2 -7410.81} C_VEL
LIN {X 0,Y 474.639,Z 414.987,A -85,B 0,C 180,E1 -7413.984,E2 -7413.984} C_VEL
LIN {X 0,Y 474.574,Z 414.995,A -85,B 0,C 180,E1 -7416.899,E2 -7416.899} C_VEL
LIN {X 0,Y 474.629,Z 414.988,A -85,B 0,C 180,E1 -7419.648,E2 -7419.648} C_VEL
LIN {X 0,Y 474.637,Z 414.988,A -85,B 0,C 180,E1 -7422.932,E2 -7422.932} C_VEL
LIN {X 0,Y 474.612,Z 414.993,A -85,B 0,C 180,E1 -7425.895,E2 -7425.895} C_VEL
LIN {X 0,Y 474.691,Z 415.134,A -85,B 0,C 180,E1 -7429.032,E2 -7429.032} C_VEL
LIN {X 0,Y 476.021,Z 423.266,A -85,B 0,C 180,E1 -7431.49,E2 -7431.49} C_VEL
LIN {X 0,Y 475.98,Z 429.464,A -85,B 0,C 180,E1 -7433.33,E2 -7433.33} C_VEL
LIN {X 0,Y 475.66,Z 441.182,A -85,B 0,C 180,E1 -7436.86,E2 -7436.86} C_VEL
LIN {X 0,Y 475.512,Z 450.931,A -85,B 0,C 180,E1 -7439.833,E2 -7439.833} C_VEL
LIN {X 0,Y 475.271,Z 460.439,A -85,B 0,C 180,E1 -7442.716,E2 -7442.716} C_VEL
LIN {X 0,Y 474.99,Z 471.41,A -85,B 0,C 180,E1 -7445.99,E2 -7445.99} C_VEL
LIN {X 0,Y 474.804,Z 481.025,A -85,B 0,C 180,E1 -7448.789,E2 -7448.789} C_VEL
LIN {X 0,Y 474.114,Z 482.63,A -85,B 0,C 180,E1 -7449.219,E2 -7449.219} C_VEL
LIN {X 0,Y 471.233,Z 485.364,A -85,B 0,C 180,E1 -7449.878,E2 -7449.878} C_VEL
LIN {X 0,Y 468.324,Z 488.126,A -85,B 0,C 180,E1 -7450.543,E2 -7450.543} C_VEL
LIN {X 0,Y 467.609,Z 489.779,A -85,B 0,C 180,E1 -7450.98,E2 -7450.98} C_VEL
LIN {X 0,Y 467.589,Z 491.36,A -85,B 0,C 180,E1 -7451.412,E2 -7451.412} C_VEL
LIN {X 0,Y 470.867,Z 506.811,A -85,B 0,C 180,E1 -7451.877,E2 -7451.877} C_VEL
LIN {X 0,Y 471.912,Z 513.074,A -85,B 0,C 180,E1 -7452.112,E2 -7452.112} C_VEL
LIN {X 0,Y 471.424,Z 526.954,A -85,B 0,C 180,E1 -7452.653,E2 -7452.653} C_VEL
LIN {X 0,Y 470.949,Z 539.698,A -85,B 0,C 180,E1 -7453.322,E2 -7453.322} C_VEL
LIN {X 0,Y 470.279,Z 552.449,A -85,B 0,C 180,E1 -7454.173,E2 -7454.173} C_VEL
LIN {X 0,Y 469.601,Z 564.189,A -85,B 0,C 180,E1 -7455.15,E2 -7455.15} C_VEL
LIN {X 0,Y 468.971,Z 573.972,A -85,B 0,C 180,E1 -7456.127,E2 -7456.127} C_VEL
LIN {X 0,Y 468.285,Z 584.927,A -85,B 0,C 180,E1 -7457.456,E2 -7457.456} C_VEL
LIN {X 0,Y 467.88,Z 593.651,A -85,B 0,C 180,E1 -7458.739,E2 -7458.739} C_VEL
LIN {X 0,Y 467.399,Z 602.166,A -85,B 0,C 180,E1 -7460.261,E2 -7460.261} C_VEL
LIN {X 0,Y 467.044,Z 609.034,A -85,B 0,C 180,E1 -7461.781,E2 -7461.781} C_VEL
LIN {X 0,Y 466.857,Z 615.114,A -85,B 0,C 180,E1 -7463.493,E2 -7463.493} C_VEL
LIN {X 0,Y 466.774,Z 618.698,A -85,B 0,C 180,E1 -7464.817,E2 -7464.817} C_VEL
LIN {X 0,Y 466.684,Z 622.118,A -85,B 0,C 180,E1 -7466.547,E2 -7466.547} C_VEL
LIN {X 0,Y 466.603,Z 624.154,A -85,B 0,C 180,E1 -7468.274,E2 -7468.274} C_VEL
LIN {X 0,Y 466.597,Z 624.858,A -85,B 0,C 180,E1 -7470,E2 -7470} C_VEL
LIN {X 0,Y 466.602,Z 624.233,A -85,B 0,C 180,E1 -7471.726,E2 -7471.726} C_VEL
LIN {X 0,Y 466.683,Z 622.263,A -85,B 0,C 180,E1 -7473.453,E2 -7473.453} C_VEL
LIN {X 0,Y 466.773,Z 618.913,A -85,B 0,C 180,E1 -7475.183,E2 -7475.183} C_VEL
LIN {X 0,Y 466.848,Z 614.083,A -85,B 0,C 180,E1 -7476.917,E2 -7476.917} C_VEL
LIN {X 0,Y 467.106,Z 607.622,A -85,B 0,C 180,E1 -7478.653,E2 -7478.653} C_VEL
LIN {X 0,Y 467.441,Z 600.422,A -85,B 0,C 180,E1 -7480.175,E2 -7480.175} C_VEL
LIN {X 0,Y 468.023,Z 591.46,A -85,B 0,C 180,E1 -7481.696,E2 -7481.696} C_VEL
LIN {X 0,Y 468.53,Z 582.083,A -85,B 0,C 180,E1 -7483.003,E2 -7483.003} C_VEL
LIN {X 0,Y 469.12,Z 571.706,A -85,B 0,C 180,E1 -7484.201,E2 -7484.201} C_VEL
LIN {X 0,Y 469.79,Z 560.26,A -85,B 0,C 180,E1 -7485.288,E2 -7485.288} C_VEL
LIN {X 0,Y 470.51,Z 547.585,A -85,B 0,C 180,E1 -7486.264,E2 -7486.264} C_VEL
LIN {X 0,Y 471.155,Z 534.452,A -85,B 0,C 180,E1 -7487.066,E2 -7487.066} C_VEL
LIN {X 0,Y 471.693,Z 520.077,A -85,B 0,C 180,E1 -7487.728,E2 -7487.728} C_VEL
LIN {X 0,Y 471.795,Z 511.565,A -85,B 0,C 180,E1 -7488.033,E2 -7488.033} C_VEL
LIN {X 0,Y 468.874,Z 497.074,A -85,B 0,C 180,E1 -7488.526,E2 -7488.526} C_VEL
LIN {X 0,Y 467.599,Z 491.305,A -85,B 0,C 180,E1 -7488.683,E2 -7488.683} C_VEL
LIN {X 0,Y 467.796,Z 480.922,A -85,B 0,C 180,E1 -7491.636,E2 -7491.636} C_VEL
LIN {X 0,Y 468,Z 469.951,A -85,B 0,C 180,E1 -7494.865,E2 -7494.865} C_VEL
LIN {X 0,Y 468.299,Z 460.46,A -85,B 0,C 180,E1 -7497.725,E2 -7497.725} C_VEL
LIN {X 0,Y 468.537,Z 450.887,A -85,B 0,C 180,E1 -7500.664,E2 -7500.664} C_VEL
LIN {X 0,Y 468.695,Z 441.034,A -85,B 0,C 180,E1 -7503.698,E2 -7503.698} C_VEL
LIN {X 0,Y 469.108,Z 428.696,A -85,B 0,C 180,E1 -7507.436,E2 -7507.436} C_VEL
LIN {X 0,Y 468.96,Z 423.495,A -85,B 0,C 180,E1 -7509.008,E2 -7509.008} C_VEL
LIN {X 0,Y 467.59,Z 415.869,A -85,B 0,C 180,E1 -7511.402,E2 -7511.402} C_VEL
LIN {X 0,Y 467.556,Z 415.871,A -85,B 0,C 180,E1 -7513.821,E2 -7513.821} C_VEL
LIN {X 0,Y 467.573,Z 415.869,A -85,B 0,C 180,E1 -7516.257,E2 -7516.257} C_VEL
LIN {X 0,Y 467.584,Z 415.871,A -85,B 0,C 180,E1 -7518.723,E2 -7518.723} C_VEL
LIN {X 0,Y 467.567,Z 415.872,A -85,B 0,C 180,E1 -7521.956,E2 -7521.956} C_VEL
LIN {X 0,Y 467.57,Z 415.87,A -85,B 0,C 180,E1 -7525.168,E2 -7525.168} C_VEL
LIN {X 0,Y 467.586,Z 415.866,A -85,B 0,C 180,E1 -7528.26,E2 -7528.26} C_VEL
LIN {X 0,Y 467.584,Z 415.867,A -85,B 0,C 180,E1 -7531.251,E2 -7531.251} C_VEL
LIN {X 0,Y 467.612,Z 415.863,A -85,B 0,C 180,E1 -7534.16,E2 -7534.16} C_VEL
LIN {X 0,Y 467.579,Z 415.866,A -85,B 0,C 180,E1 -7536.996,E2 -7536.996} C_VEL
LIN {X 0,Y 467.628,Z 415.862,A -85,B 0,C 180,E1 -7539.418,E2 -7539.418} C_VEL
LIN {X 0,Y 472.563,Z 431.238,A -85,B 0,C 180,E1 -7540.334,E2 -7540.334} C_VEL
LIN {X 0,Y 472.016,Z 444.828,A -85,B 0,C 180,E1 -7541.104,E2 -7541.104} C_VEL
LIN {X 0,Y 471.248,Z 458.796,A -85,B 0,C 180,E1 -7542.086,E2 -7542.086} C_VEL
LIN {X 0,Y 470.524,Z 471.45,A -85,B 0,C 180,E1 -7543.175,E2 -7543.175} C_VEL
LIN {X 0,Y 469.802,Z 483.094,A -85,B 0,C 180,E1 -7544.379,E2 -7544.379} C_VEL
LIN {X 0,Y 469.161,Z 493.71,A -85,B 0,C 180,E1 -7545.69,E2 -7545.69} C_VEL
LIN {X 0,Y 468.438,Z 504.025,A -85,B 0,C 180,E1 -7547.213,E2 -7547.213} C_VEL
LIN {X 0,Y 467.995,Z 512.576,A -85,B 0,C 180,E1 -7548.742,E2 -7548.742} C_VEL
LIN {X 0,Y 467.545,Z 520.556,A -85,B 0,C 180,E1 -7550.482,E2 -7550.482} C_VEL
LIN {X 0,Y 467.262,Z 526.898,A -85,B 0,C 180,E1 -7552.22,E2 -7552.22} C_VEL
LIN {X 0,Y 467.042,Z 531.811,A -85,B 0,C 180,E1 -7553.953,E2 -7553.953} C_VEL
LIN {X 0,Y 467.017,Z 535.417,A -85,B 0,C 180,E1 -7555.685,E2 -7555.685} C_VEL
LIN {X 0,Y 466.847,Z 537.839,A -85,B 0,C 180,E1 -7557.411,E2 -7557.411} C_VEL
LIN {X 0,Y 466.724,Z 539.115,A -85,B 0,C 180,E1 -7559.137,E2 -7559.137} C_VEL
LIN {X 0,Y 466.729,Z 539.214,A -85,B 0,C 180,E1 -7560.863,E2 -7560.863} C_VEL
LIN {X 0,Y 466.864,Z 538.155,A -85,B 0,C 180,E1 -7562.588,E2 -7562.588} C_VEL
LIN {X 0,Y 467.054,Z 535.948,A -85,B 0,C 180,E1 -7564.315,E2 -7564.315} C_VEL
LIN {X 0,Y 467.173,Z 532.557,A -85,B 0,C 180,E1 -7566.045,E2 -7566.045} C_VEL
LIN {X 0,Y 467.339,Z 527.87,A -85,B 0,C 180,E1 -7567.779,E2 -7567.779} C_VEL
LIN {X 0,Y 467.618,Z 521.735,A -85,B 0,C 180,E1 -7569.516,E2 -7569.516} C_VEL
LIN {X 0,Y 468.09,Z 513.953,A -85,B 0,C 180,E1 -7571.255,E2 -7571.255} C_VEL
LIN {X 0,Y 468.6,Z 505.008,A -85,B 0,C 180,E1 -7572.874,E2 -7572.874} C_VEL
LIN {X 0,Y 469.244,Z 495.364,A -85,B 0,C 180,E1 -7574.307,E2 -7574.307} C_VEL
LIN {X 0,Y 469.855,Z 484.834,A -85,B 0,C 180,E1 -7575.619,E2 -7575.619} C_VEL
LIN {X 0,Y 470.505,Z 473.096,A -85,B 0,C 180,E1 -7576.838,E2 -7576.838} C_VEL
LIN {X 0,Y 471.256,Z 460.501,A -85,B 0,C 180,E1 -7577.914,E2 -7577.914} C_VEL
LIN {X 0,Y 471.855,Z 448.06,A -85,B 0,C 180,E1 -7578.789,E2 -7578.789} C_VEL
LIN {X 0,Y 472.465,Z 433.488,A -85,B 0,C 180,E1 -7579.611,E2 -7579.611} C_VEL
LIN {X 0,Y 472.439,Z 430.931,A -85,B 0,C 180,E1 -7579.744,E2 -7579.744} C_VEL
LIN {X 0,Y 468.233,Z 417.991,A -85,B 0,C 180,E1 -7580.501,E2 -7580.501} C_VEL
LIN {X 0,Y 467.628,Z 415.863,A -85,B 0,C 180,E1 -7580.625,E2 -7580.625} C_VEL
LIN {X 0,Y 467.565,Z 415.872,A -85,B 0,C 180,E1 -7583.944,E2 -7583.944} C_VEL
LIN {X 0,Y 467.614,Z 415.863,A -85,B 0,C 180,E1 -7586.8,E2 -7586.8} C_VEL
LIN {X 0,Y 467.556,Z 415.873,A -85,B 0,C 180,E1 -7589.738,E2 -7589.738} C_VEL
LIN {X 0,Y 467.585,Z 415.864,A -85,B 0,C 180,E1 -7592.758,E2 -7592.758} C_VEL
LIN {X 0,Y 467.555,Z 415.872,A -85,B 0,C 180,E1 -7595.89,E2 -7595.89} C_VEL
LIN {X 0,Y 467.583,Z 415.867,A -85,B 0,C 180,E1 -7599.145,E2 -7599.145} C_VEL
LIN {X 0,Y 467.587,Z 415.868,A -85,B 0,C 180,E1 -7602.567,E2 -7602.567} C_VEL
LIN {X 0,Y 467.641,Z 415.947,A -85,B 0,C 180,E1 -7603.66,E2 -7603.66} C_VEL
LIN {X 0,Y 467.934,Z 419.474,A -85,B 0,C 180,E1 -7605.097,E2 -7605.097} C_VEL
LIN {X 0,Y 467.515,Z 430.959,A -85,B 0,C 180,E1 -7609.237,E2 -7609.237} C_VEL
LIN {X 0,Y 467.658,Z 440.418,A -85,B 0,C 180,E1 -7612.413,E2 -7612.413} C_VEL
LIN {X 0,Y 467.781,Z 450.638,A -85,B 0,C 180,E1 -7615.723,E2 -7615.723} C_VEL
LIN {X 0,Y 467.787,Z 460.668,A -85,B 0,C 180,E1 -7618.911,E2 -7618.911} C_VEL
LIN {X 0,Y 467.769,Z 469.686,A -85,B 0,C 180,E1 -7621.753,E2 -7621.753} C_VEL
LIN {X 0,Y 467.609,Z 479.209,A -85,B 0,C 180,E1 -7624.75,E2 -7624.75} C_VEL
LIN {X 0,Y 467.492,Z 489.215,A -85,B 0,C 180,E1 -7627.924,E2 -7627.924} C_VEL
LIN {X 0,Y 467.291,Z 499.084,A -85,B 0,C 180,E1 -7631.069,E2 -7631.069} C_VEL
LIN {X 0,Y 467.298,Z 499.775,A -85,B 0,C 180,E1 -7631.289,E2 -7631.289} C_VEL
LIN {X 0,Y 468.288,Z 506.495,A -85,B 0,C 180,E1 -7631.473,E2 -7631.473} C_VEL
LIN {X 0,Y 471.412,Z 521.69,A -85,B 0,C 180,E1 -7632.033,E2 -7632.033} C_VEL
LIN {X 0,Y 471.792,Z 525.166,A -85,B 0,C 180,E1 -7632.172,E2 -7632.172} C_VEL
LIN {X 0,Y 471.286,Z 538.136,A -85,B 0,C 180,E1 -7632.725,E2 -7632.725} C_VEL
LIN {X 0,Y 470.61,Z 552.291,A -85,B 0,C 180,E1 -7633.516,E2 -7633.516} C_VEL
LIN {X 0,Y 469.881,Z 565.953,A -85,B 0,C 180,E1 -7634.493,E2 -7634.493} C_VEL
LIN {X 0,Y 469.177,Z 578.215,A -85,B 0,C 180,E1 -7635.58,E2 -7635.58} C_VEL
LIN {X 0,Y 468.557,Z 589.292,A -85,B 0,C 180,E1 -7636.777,E2 -7636.777} C_VEL
LIN {X 0,Y 468.081,Z 599.252,A -85,B 0,C 180,E1 -7638.086,E2 -7638.086} C_VEL
LIN {X 0,Y 467.581,Z 607.416,A -85,B 0,C 180,E1 -7639.39,E2 -7639.39} C_VEL
LIN {X 0,Y 467.183,Z 615.129,A -85,B 0,C 180,E1 -7640.912,E2 -7640.912} C_VEL
LIN {X 0,Y 466.929,Z 620.545,A -85,B 0,C 180,E1 -7642.215,E2 -7642.215} C_VEL
LIN {X 0,Y 466.771,Z 626.201,A -85,B 0,C 180,E1 -7643.95,E2 -7643.95} C_VEL
LIN {X 0,Y 466.764,Z 628.439,A -85,B 0,C 180,E1 -7644.817,E2 -7644.817} C_VEL
LIN {X 0,Y 466.681,Z 631.824,A -85,B 0,C 180,E1 -7646.547,E2 -7646.547} C_VEL
LIN {X 0,Y 466.601,Z 633.83,A -85,B 0,C 180,E1 -7648.274,E2 -7648.274} C_VEL
LIN {X 0,Y 466.568,Z 634.5,A -85,B 0,C 180,E1 -7650,E2 -7650} C_VEL
LIN {X 0,Y 466.601,Z 633.827,A -85,B 0,C 180,E1 -7651.726,E2 -7651.726} C_VEL
LIN {X 0,Y 466.681,Z 631.824,A -85,B 0,C 180,E1 -7653.453,E2 -7653.453} C_VEL
LIN {X 0,Y 466.763,Z 628.443,A -85,B 0,C 180,E1 -7655.183,E2 -7655.183} C_VEL
LIN {X 0,Y 466.832,Z 623.598,A -85,B 0,C 180,E1 -7656.917,E2 -7656.917} C_VEL
LIN {X 0,Y 467.032,Z 618.856,A -85,B 0,C 180,E1 -7658.219,E2 -7658.219} C_VEL
LIN {X 0,Y 467.374,Z 612.054,A -85,B 0,C 180,E1 -7659.739,E2 -7659.739} C_VEL
LIN {X 0,Y 467.744,Z 604.887,A -85,B 0,C 180,E1 -7661.045,E2 -7661.045} C_VEL
LIN {X 0,Y 468.212,Z 596.373,A -85,B 0,C 180,E1 -7662.324,E2 -7662.324} C_VEL
LIN {X 0,Y 468.808,Z 585.603,A -85,B 0,C 180,E1 -7663.657,E2 -7663.657} C_VEL
LIN {X 0,Y 469.421,Z 573.831,A -85,B 0,C 180,E1 -7664.856,E2 -7664.856} C_VEL
LIN {X 0,Y 470.178,Z 562.131,A -85,B 0,C 180,E1 -7665.831,E2 -7665.831} C_VEL
LIN {X 0,Y 470.812,Z 549.631,A -85,B 0,C 180,E1 -7666.679,E2 -7666.679} C_VEL
LIN {X 0,Y 471.421,Z 535.559,A -85,B 0,C 180,E1 -7667.423,E2 -7667.423} C_VEL
LIN {X 0,Y 471.707,Z 523.043,A -85,B 0,C 180,E1 -7667.931,E2 -7667.931} C_VEL
LIN {X 0,Y 468.705,Z 508.204,A -85,B 0,C 180,E1 -7668.486,E2 -7668.486} C_VEL
LIN {X 0,Y 467.288,Z 501.093,A -85,B 0,C 180,E1 -7668.704,E2 -7668.704} C_VEL
LIN {X 0,Y 467.491,Z 492.814,A -85,B 0,C 180,E1 -7671.612,E2 -7671.612} C_VEL
LIN {X 0,Y 467.719,Z 483.563,A -85,B 0,C 180,E1 -7674.881,E2 -7674.881} C_VEL
LIN {X 0,Y 467.981,Z 474.349,A -85,B 0,C 180,E1 -7678.233,E2 -7678.233} C_VEL
LIN {X 0,Y 468.218,Z 466.479,A -85,B 0,C 180,E1 -7681.176,E2 -7681.176} C_VEL
LIN {X 0,Y 468.416,Z 459.841,A -85,B 0,C 180,E1 -7683.72,E2 -7683.72} C_VEL
LIN {X 0,Y 468.679,Z 451.901,A -85,B 0,C 180,E1 -7686.857,E2 -7686.857} C_VEL
LIN {X 0,Y 468.941,Z 443.84,A -85,B 0,C 180,E1 -7690.152,E2 -7690.152} C_VEL
LIN {X 0,Y 469.163,Z 437.62,A -85,B 0,C 180,E1 -7692.776,E2 -7692.776} C_VEL
LIN {X 0,Y 469.549,Z 430.376,A -85,B 0,C 180,E1 -7695.926,E2 -7695.926} C_VEL
LIN {X 0,Y 469.419,Z 426.618,A -85,B 0,C 180,E1 -7697.645,E2 -7697.645} C_VEL
LIN {X 0,Y 468.482,Z 420.889,A -85,B 0,C 180,E1 -7700.412,E2 -7700.412} C_VEL
LIN {X 0,Y 467.554,Z 415.871,A -85,B 0,C 180,E1 -7703.04,E2 -7703.04} C_VEL
LIN {X 0,Y 467.588,Z 415.865,A -85,B 0,C 180,E1 -7706.212,E2 -7706.212} C_VEL
LIN {X 0,Y 467.571,Z 415.868,A -85,B 0,C 180,E1 -7709.266,E2 -7709.266} C_VEL
LIN {X 0,Y 467.646,Z 415.858,A -85,B 0,C 180,E1 -7712.459,E2 -7712.459} C_VEL
LIN {X 0,Y 467.606,Z 415.86,A -85,B 0,C 180,E1 -7715.113,E2 -7715.113} C_VEL
LIN {X 0,Y 467.538,Z 415.868,A -85,B 0,C 180,E1 -7717.926,E2 -7717.926} C_VEL
LIN {X 0,Y 467.626,Z 415.861,A -85,B 0,C 180,E1 -7720.692,E2 -7720.692} C_VEL
LIN {X 0,Y 467.652,Z 415.852,A -85,B 0,C 180,E1 -7724.115,E2 -7724.115} C_VEL
LIN {X 0,Y 467.656,Z 415.857,A -85,B 0,C 180,E1 -7727.642,E2 -7727.642} C_VEL
LIN {X 0,Y 467.664,Z 415.85,A -85,B 0,C 180,E1 -7730.485,E2 -7730.485} C_VEL
LIN {X 0,Y 467.701,Z 415.85,A -85,B 0,C 180,E1 -7733.096,E2 -7733.096} C_VEL
LIN {X 0,Y 467.727,Z 415.847,A -85,B 0,C 180,E1 -7734.828,E2 -7734.828} C_VEL
LIN {X 0,Y 467.862,Z 415.825,A -85,B 0,C 180,E1 -7737.417,E2 -7737.417} C_VEL
LIN {X 0,Y 467.885,Z 415.832,A -85,B 0,C 180,E1 -7740,E2 -7740} C_VEL
LIN {X 0,Y 467.861,Z 415.826,A -85,B 0,C 180,E1 -7742.583,E2 -7742.583} C_VEL
LIN {X 0,Y 467.746,Z 415.849,A -85,B 0,C 180,E1 -7746.037,E2 -7746.037} C_VEL
LIN {X 0,Y 467.684,Z 415.846,A -85,B 0,C 180,E1 -7748.643,E2 -7748.643} C_VEL
LIN {X 0,Y 467.658,Z 415.857,A -85,B 0,C 180,E1 -7752.145,E2 -7752.145} C_VEL
LIN {X 0,Y 467.642,Z 415.858,A -85,B 0,C 180,E1 -7755.695,E2 -7755.695} C_VEL
LIN {X 0,Y 467.62,Z 415.855,A -85,B 0,C 180,E1 -7758.765,E2 -7758.765} C_VEL
LIN {X 0,Y 467.583,Z 415.867,A -85,B 0,C 180,E1 -7761.268,E2 -7761.268} C_VEL
LIN {X 0,Y 467.565,Z 415.867,A -85,B 0,C 180,E1 -7763.944,E2 -7763.944} C_VEL
LIN {X 0,Y 467.615,Z 415.859,A -85,B 0,C 180,E1 -7766.801,E2 -7766.801} C_VEL
LIN {X 0,Y 467.556,Z 415.869,A -85,B 0,C 180,E1 -7769.738,E2 -7769.738} C_VEL
LIN {X 0,Y 467.585,Z 415.866,A -85,B 0,C 180,E1 -7772.758,E2 -7772.758} C_VEL
LIN {X 0,Y 467.555,Z 415.869,A -85,B 0,C 180,E1 -7775.89,E2 -7775.89} C_VEL
LIN {X 0,Y 467.584,Z 415.869,A -85,B 0,C 180,E1 -7779.145,E2 -7779.145} C_VEL
LIN {X 0,Y 467.588,Z 415.867,A -85,B 0,C 180,E1 -7782.567,E2 -7782.567} C_VEL
LIN {X 0,Y 467.573,Z 415.871,A -85,B 0,C 180,E1 -7785.053,E2 -7785.053} C_VEL
LIN {X 0,Y 467.598,Z 415.872,A -85,B 0,C 180,E1 -7788.599,E2 -7788.599} C_VEL
LIN {X 0,Y 467.633,Z 416.019,A -85,B 0,C 180,E1 -7788.797,E2 -7788.797} C_VEL
LIN {X 0,Y 468.995,Z 423.829,A -85,B 0,C 180,E1 -7791.191,E2 -7791.191} C_VEL
LIN {X 0,Y 469.092,Z 429.406,A -85,B 0,C 180,E1 -7792.872,E2 -7792.872} C_VEL
LIN {X 0,Y 468.695,Z 442.187,A -85,B 0,C 180,E1 -7796.758,E2 -7796.758} C_VEL
LIN {X 0,Y 468.505,Z 452.182,A -85,B 0,C 180,E1 -7799.832,E2 -7799.832} C_VEL
LIN {X 0,Y 468.253,Z 461.79,A -85,B 0,C 180,E1 -7802.772,E2 -7802.772} C_VEL
LIN {X 0,Y 467.966,Z 472.799,A -85,B 0,C 180,E1 -7806.078,E2 -7806.078} C_VEL
LIN {X 0,Y 467.726,Z 483.914,A -85,B 0,C 180,E1 -7809.322,E2 -7809.322} C_VEL
LIN {X 0,Y 467.609,Z 489.779,A -85,B 0,C 180,E1 -7810.98,E2 -7810.98} C_VEL
LIN {X 0,Y 467.825,Z 491.655,A -85,B 0,C 180,E1 -7811.265,E2 -7811.265} C_VEL
LIN {X 0,Y 468.264,Z 495.304,A -85,B 0,C 180,E1 -7811.491,E2 -7811.491} C_VEL
LIN {X 0,Y 467.847,Z 500.757,A -85,B 0,C 180,E1 -7811.601,E2 -7811.601} C_VEL
LIN {X 0,Y 465.504,Z 515.84,A -85,B 0,C 180,E1 -7811.941,E2 -7811.941} C_VEL
LIN {X 0,Y 464.894,Z 520.11,A -85,B 0,C 180,E1 -7812.096,E2 -7812.096} C_VEL
LIN {X 0,Y 464.382,Z 532.98,A -85,B 0,C 180,E1 -7812.688,E2 -7812.688} C_VEL
LIN {X 0,Y 463.768,Z 546.379,A -85,B 0,C 180,E1 -7813.493,E2 -7813.493} C_VEL
LIN {X 0,Y 462.923,Z 559.292,A -85,B 0,C 180,E1 -7814.48,E2 -7814.48} C_VEL
LIN {X 0,Y 462.275,Z 570.908,A -85,B 0,C 180,E1 -7815.585,E2 -7815.585} C_VEL
LIN {X 0,Y 461.595,Z 581.427,A -85,B 0,C 180,E1 -7816.798,E2 -7816.798} C_VEL
LIN {X 0,Y 461.075,Z 590.919,A -85,B 0,C 180,E1 -7818.125,E2 -7818.125} C_VEL
LIN {X 0,Y 460.509,Z 598.796,A -85,B 0,C 180,E1 -7819.447,E2 -7819.447} C_VEL
LIN {X 0,Y 460.178,Z 605.352,A -85,B 0,C 180,E1 -7820.772,E2 -7820.772} C_VEL
LIN {X 0,Y 459.904,Z 610.796,A -85,B 0,C 180,E1 -7822.095,E2 -7822.095} C_VEL
LIN {X 0,Y 459.724,Z 616.496,A -85,B 0,C 180,E1 -7823.857,E2 -7823.857} C_VEL
LIN {X 0,Y 459.71,Z 618.756,A -85,B 0,C 180,E1 -7824.737,E2 -7824.737} C_VEL
LIN {X 0,Y 459.581,Z 622.177,A -85,B 0,C 180,E1 -7826.493,E2 -7826.493} C_VEL
LIN {X 0,Y 459.515,Z 624.213,A -85,B 0,C 180,E1 -7828.247,E2 -7828.247} C_VEL
LIN {X 0,Y 459.5,Z 624.916,A -85,B 0,C 180,E1 -7830,E2 -7830} C_VEL
LIN {X 0,Y 459.514,Z 624.29,A -85,B 0,C 180,E1 -7831.753,E2 -7831.753} C_VEL
LIN {X 0,Y 459.58,Z 622.32,A -85,B 0,C 180,E1 -7833.507,E2 -7833.507} C_VEL
LIN {X 0,Y 459.709,Z 618.968,A -85,B 0,C 180,E1 -7835.263,E2 -7835.263} C_VEL
LIN {X 0,Y 459.769,Z 614.137,A -85,B 0,C 180,E1 -7837.024,E2 -7837.024} C_VEL
LIN {X 0,Y 460.065,Z 607.675,A -85,B 0,C 180,E1 -7838.787,E2 -7838.787} C_VEL
LIN {X 0,Y 460.425,Z 600.474,A -85,B 0,C 180,E1 -7840.332,E2 -7840.332} C_VEL
LIN {X 0,Y 461.047,Z 591.509,A -85,B 0,C 180,E1 -7841.876,E2 -7841.876} C_VEL
LIN {X 0,Y 461.59,Z 582.13,A -85,B 0,C 180,E1 -7843.202,E2 -7843.202} C_VEL
LIN {X 0,Y 462.205,Z 571.75,A -85,B 0,C 180,E1 -7844.418,E2 -7844.418} C_VEL
LIN {X 0,Y 462.904,Z 560.3,A -85,B 0,C 180,E1 -7845.521,E2 -7845.521} C_VEL
LIN {X 0,Y 463.694,Z 547.619,A -85,B 0,C 180,E1 -7846.51,E2 -7846.51} C_VEL
LIN {X 0,Y 464.347,Z 535.065,A -85,B 0,C 180,E1 -7847.29,E2 -7847.29} C_VEL
LIN {X 0,Y 464.891,Z 521.079,A -85,B 0,C 180,E1 -7847.957,E2 -7847.957} C_VEL
LIN {X 0,Y 464.951,Z 512.38,A -85,B 0,C 180,E1 -7848.28,E2 -7848.28} C_VEL
LIN {X 0,Y 462.06,Z 497.953,A -85,B 0,C 180,E1 -7848.789,E2 -7848.789} C_VEL
LIN {X 0,Y 460.596,Z 491.26,A -85,B 0,C 180,E1 -7848.985,E2 -7848.985} C_VEL
LIN {X 0,Y 460.81,Z 479.312,A -85,B 0,C 180,E1 -7852.413,E2 -7852.413} C_VEL
LIN {X 0,Y 461.057,Z 468.639,A -85,B 0,C 180,E1 -7855.601,E2 -7855.601} C_VEL
LIN {X 0,Y 461.33,Z 460.179,A -85,B 0,C 180,E1 -7858.181,E2 -7858.181} C_VEL
LIN {X 0,Y 461.572,Z 449.481,A -85,B 0,C 180,E1 -7861.497,E2 -7861.497} C_VEL
LIN {X 0,Y 461.776,Z 440.549,A -85,B 0,C 180,E1 -7864.272,E2 -7864.272} C_VEL
LIN {X 0,Y 462.198,Z 429.18,A -85,B 0,C 180,E1 -7867.75,E2 -7867.75} C_VEL
LIN {X 0,Y 461.858,Z 423.891,A -85,B 0,C 180,E1 -7869.377,E2 -7869.377} C_VEL
LIN {X 0,Y 460.543,Z 416.747,A -85,B 0,C 180,E1 -7871.604,E2 -7871.604} C_VEL
LIN {X 0,Y 460.519,Z 416.748,A -85,B 0,C 180,E1 -7874.588,E2 -7874.588} C_VEL
LIN {X 0,Y 460.526,Z 416.751,A -85,B 0,C 180,E1 -7877.819,E2 -7877.819} C_VEL
LIN {X 0,Y 460.546,Z 416.746,A -85,B 0,C 180,E1 -7881.102,E2 -7881.102} C_VEL
LIN {X 0,Y 460.515,Z 416.748,A -85,B 0,C 180,E1 -7884.555,E2 -7884.555} C_VEL
LIN {X 0,Y 460.534,Z 416.747,A -85,B 0,C 180,E1 -7887.716,E2 -7887.716} C_VEL
LIN {X 0,Y 460.549,Z 416.742,A -85,B 0,C 180,E1 -7890.77,E2 -7890.77} C_VEL
LIN {X 0,Y 460.565,Z 416.743,A -85,B 0,C 180,E1 -7893.735,E2 -7893.735} C_VEL
LIN {X 0,Y 460.548,Z 416.742,A -85,B 0,C 180,E1 -7896.624,E2 -7896.624} C_VEL
LIN {X 0,Y 460.59,Z 416.854,A -85,B 0,C 180,E1 -7899.148,E2 -7899.148} C_VEL
LIN {X 0,Y 465.236,Z 431.094,A -85,B 0,C 180,E1 -7900.009,E2 -7900.009} C_VEL
LIN {X 0,Y 465.798,Z 433.546,A -85,B 0,C 180,E1 -7900.162,E2 -7900.162} C_VEL
LIN {X 0,Y 465.077,Z 448.359,A -85,B 0,C 180,E1 -7901.041,E2 -7901.041} C_VEL
LIN {X 0,Y 464.331,Z 461.788,A -85,B 0,C 180,E1 -7902.038,E2 -7902.038} C_VEL
LIN {X 0,Y 463.472,Z 475.188,A -85,B 0,C 180,E1 -7903.255,E2 -7903.255} C_VEL
LIN {X 0,Y 462.699,Z 487.242,A -85,B 0,C 180,E1 -7904.585,E2 -7904.585} C_VEL
LIN {X 0,Y 462.021,Z 497.354,A -85,B 0,C 180,E1 -7905.914,E2 -7905.914} C_VEL
LIN {X 0,Y 461.39,Z 507.361,A -85,B 0,C 180,E1 -7907.496,E2 -7907.496} C_VEL
LIN {X 0,Y 460.899,Z 515.348,A -85,B 0,C 180,E1 -7909.012,E2 -7909.012} C_VEL
LIN {X 0,Y 460.494,Z 522.931,A -85,B 0,C 180,E1 -7910.779,E2 -7910.779} C_VEL
LIN {X 0,Y 460.192,Z 528.946,A -85,B 0,C 180,E1 -7912.541,E2 -7912.541} C_VEL
LIN {X 0,Y 460.003,Z 532.497,A -85,B 0,C 180,E1 -7913.861,E2 -7913.861} C_VEL
LIN {X 0,Y 459.977,Z 536.134,A -85,B 0,C 180,E1 -7915.619,E2 -7915.619} C_VEL
LIN {X 0,Y 459.793,Z 538.58,A -85,B 0,C 180,E1 -7917.372,E2 -7917.372} C_VEL
LIN {X 0,Y 459.665,Z 539.872,A -85,B 0,C 180,E1 -7919.124,E2 -7919.124} C_VEL
LIN {X 0,Y 459.673,Z 539.986,A -85,B 0,C 180,E1 -7920.876,E2 -7920.876} C_VEL
LIN {X 0,Y 459.812,Z 538.934,A -85,B 0,C 180,E1 -7922.628,E2 -7922.628} C_VEL
LIN {X 0,Y 460.03,Z 536.731,A -85,B 0,C 180,E1 -7924.381,E2 -7924.381} C_VEL
LIN {X 0,Y 460.153,Z 533.339,A -85,B 0,C 180,E1 -7926.137,E2 -7926.137} C_VEL
LIN {X 0,Y 460.355,Z 528.638,A -85,B 0,C 180,E1 -7927.897,E2 -7927.897} C_VEL
LIN {X 0,Y 460.642,Z 522.484,A -85,B 0,C 180,E1 -7929.661,E2 -7929.661} C_VEL
LIN {X 0,Y 461.156,Z 514.668,A -85,B 0,C 180,E1 -7931.427,E2 -7931.427} C_VEL
LIN {X 0,Y 461.683,Z 505.947,A -85,B 0,C 180,E1 -7933.032,E2 -7933.032} C_VEL
LIN {X 0,Y 462.393,Z 496.066,A -85,B 0,C 180,E1 -7934.524,E2 -7934.524} C_VEL
LIN {X 0,Y 463.035,Z 485.493,A -85,B 0,C 180,E1 -7935.855,E2 -7935.855} C_VEL
LIN {X 0,Y 463.698,Z 474.06,A -85,B 0,C 180,E1 -7937.056,E2 -7937.056} C_VEL
LIN {X 0,Y 464.459,Z 462.398,A -85,B 0,C 180,E1 -7938.071,E2 -7938.071} C_VEL
LIN {X 0,Y 465.079,Z 450.238,A -85,B 0,C 180,E1 -7938.959,E2 -7938.959} C_VEL
LIN {X 0,Y 465.68,Z 436.432,A -85,B 0,C 180,E1 -7939.775,E2 -7939.775} C_VEL
LIN {X 0,Y 465.6,Z 432.078,A -85,B 0,C 180,E1 -7940.01,E2 -7940.01} C_VEL
LIN {X 0,Y 460.982,Z 418.345,A -85,B 0,C 180,E1 -7940.839,E2 -7940.839} C_VEL
LIN {X 0,Y 460.571,Z 416.741,A -85,B 0,C 180,E1 -7940.926,E2 -7940.926} C_VEL
LIN {X 0,Y 460.532,Z 416.748,A -85,B 0,C 180,E1 -7944.333,E2 -7944.333} C_VEL
LIN {X 0,Y 460.59,Z 416.742,A -85,B 0,C 180,E1 -7947.748,E2 -7947.748} C_VEL
LIN {X 0,Y 460.524,Z 416.745,A -85,B 0,C 180,E1 -7951.283,E2 -7951.283} C_VEL
LIN {X 0,Y 460.533,Z 416.743,A -85,B 0,C 180,E1 -7954.505,E2 -7954.505} C_VEL
LIN {X 0,Y 460.502,Z 416.751,A -85,B 0,C 180,E1 -7957.623,E2 -7957.623} C_VEL
LIN {X 0,Y 460.544,Z 416.743,A -85,B 0,C 180,E1 -7960.27,E2 -7960.27} C_VEL
LIN {X 0,Y 460.609,Z 416.786,A -85,B 0,C 180,E1 -7963.438,E2 -7963.438} C_VEL
LIN {X 0,Y 460.937,Z 420.495,A -85,B 0,C 180,E1 -7965.005,E2 -7965.005} C_VEL
LIN {X 0,Y 460.461,Z 431.194,A -85,B 0,C 180,E1 -7968.981,E2 -7968.981} C_VEL
LIN {X 0,Y 460.572,Z 439.421,A -85,B 0,C 180,E1 -7971.83,E2 -7971.83} C_VEL
LIN {X 0,Y 460.71,Z 449.11,A -85,B 0,C 180,E1 -7975.054,E2 -7975.054} C_VEL
LIN {X 0,Y 460.711,Z 458.92,A -85,B 0,C 180,E1 -7978.242,E2 -7978.242} C_VEL
LIN {X 0,Y 460.719,Z 468.38,A -85,B 0,C 180,E1 -7981.281,E2 -7981.281} C_VEL
LIN {X 0,Y 460.538,Z 479.072,A -85,B 0,C 180,E1 -7984.704,E2 -7984.704} C_VEL
LIN {X 0,Y 460.389,Z 489.453,A -85,B 0,C 180,E1 -7988.037,E2 -7988.037} C_VEL
LIN {X 0,Y 460.221,Z 498.492,A -85,B 0,C 180,E1 -7990.961,E2 -7990.961} C_VEL
LIN {X 0,Y 461.757,Z 508.624,A -85,B 0,C 180,E1 -7991.259,E2 -7991.259} C_VEL
LIN {X 0,Y 464.766,Z 523.797,A -85,B 0,C 180,E1 -7991.87,E2 -7991.87} C_VEL
LIN {X 0,Y 464.77,Z 528.343,A -85,B 0,C 180,E1 -7992.055,E2 -7992.055} C_VEL
LIN {X 0,Y 464.251,Z 541.795,A -85,B 0,C 180,E1 -7992.7,E2 -7992.7} C_VEL
LIN {X 0,Y 463.54,Z 554.645,A -85,B 0,C 180,E1 -7993.484,E2 -7993.484} C_VEL
LIN {X 0,Y 462.782,Z 567.64,A -85,B 0,C 180,E1 -7994.475,E2 -7994.475} C_VEL
LIN {X 0,Y 462.098,Z 579.4,A -85,B 0,C 180,E1 -7995.579,E2 -7995.579} C_VEL
LIN {X 0,Y 461.453,Z 590.103,A -85,B 0,C 180,E1 -7996.794,E2 -7996.794} C_VEL
LIN {X 0,Y 460.974,Z 599.81,A -85,B 0,C 180,E1 -7998.122,E2 -7998.122} C_VEL
LIN {X 0,Y 460.371,Z 609.085,A -85,B 0,C 180,E1 -7999.667,E2 -7999.667} C_VEL
LIN {X 0,Y 460.028,Z 616.594,A -85,B 0,C 180,E1 -8001.212,E2 -8001.212} C_VEL
LIN {X 0,Y 459.794,Z 621.79,A -85,B 0,C 180,E1 -8002.535,E2 -8002.535} C_VEL
LIN {X 0,Y 459.679,Z 627.257,A -85,B 0,C 180,E1 -8004.297,E2 -8004.297} C_VEL
LIN {X 0,Y 459.559,Z 630.243,A -85,B 0,C 180,E1 -8005.615,E2 -8005.615} C_VEL
LIN {X 0,Y 459.566,Z 632.978,A -85,B 0,C 180,E1 -8007.37,E2 -8007.37} C_VEL
LIN {X 0,Y 459.492,Z 634.326,A -85,B 0,C 180,E1 -8009.124,E2 -8009.124} C_VEL
LIN {X 0,Y 459.492,Z 634.324,A -85,B 0,C 180,E1 -8010.876,E2 -8010.876} C_VEL
LIN {X 0,Y 459.566,Z 632.976,A -85,B 0,C 180,E1 -8012.63,E2 -8012.63} C_VEL
LIN {X 0,Y 459.558,Z 630.244,A -85,B 0,C 180,E1 -8014.385,E2 -8014.385} C_VEL
LIN {X 0,Y 459.676,Z 627.239,A -85,B 0,C 180,E1 -8015.703,E2 -8015.703} C_VEL
LIN {X 0,Y 459.794,Z 621.823,A -85,B 0,C 180,E1 -8017.465,E2 -8017.465} C_VEL
LIN {X 0,Y 460.032,Z 616.655,A -85,B 0,C 180,E1 -8018.788,E2 -8018.788} C_VEL
LIN {X 0,Y 460.406,Z 609.219,A -85,B 0,C 180,E1 -8020.333,E2 -8020.333} C_VEL
LIN {X 0,Y 460.969,Z 600.086,A -85,B 0,C 180,E1 -8021.878,E2 -8021.878} C_VEL
LIN {X 0,Y 461.508,Z 590.507,A -85,B 0,C 180,E1 -8023.204,E2 -8023.204} C_VEL
LIN {X 0,Y 462.221,Z 578.851,A -85,B 0,C 180,E1 -8024.53,E2 -8024.53} C_VEL
LIN {X 0,Y 462.906,Z 567.025,A -85,B 0,C 180,E1 -8025.634,E2 -8025.634} C_VEL
LIN {X 0,Y 463.724,Z 553.906,A -85,B 0,C 180,E1 -8026.622,E2 -8026.622} C_VEL
LIN {X 0,Y 464.398,Z 540.527,A -85,B 0,C 180,E1 -8027.418,E2 -8027.418} C_VEL
LIN {X 0,Y 464.981,Z 526.678,A -85,B 0,C 180,E1 -8028.05,E2 -8028.05} C_VEL
LIN {X 0,Y 464.735,Z 523.029,A -85,B 0,C 180,E1 -8028.202,E2 -8028.202} C_VEL
LIN {X 0,Y 461.647,Z 508.06,A -85,B 0,C 180,E1 -8028.786,E2 -8028.786} C_VEL
LIN {X 0,Y 460.215,Z 500.431,A -85,B 0,C 180,E1 -8029.023,E2 -8029.023} C_VEL
LIN {X 0,Y 460.463,Z 490.885,A -85,B 0,C 180,E1 -8032.431,E2 -8032.431} C_VEL
LIN {X 0,Y 460.702,Z 483.026,A -85,B 0,C 180,E1 -8035.286,E2 -8035.286} C_VEL
LIN {X 0,Y 460.996,Z 473.822,A -85,B 0,C 180,E1 -8038.7,E2 -8038.7} C_VEL
LIN {X 0,Y 461.288,Z 464.625,A -85,B 0,C 180,E1 -8042.225,E2 -8042.225} C_VEL
LIN {X 0,Y 461.533,Z 456.702,A -85,B 0,C 180,E1 -8045.355,E2 -8045.355} C_VEL
LIN {X 0,Y 461.775,Z 448.724,A -85,B 0,C 180,E1 -8048.609,E2 -8048.609} C_VEL
LIN {X 0,Y 462.079,Z 441.105,A -85,B 0,C 180,E1 -8051.818,E2 -8051.818} C_VEL
LIN {X 0,Y 462.469,Z 433.878,A -85,B 0,C 180,E1 -8054.962,E2 -8054.962} C_VEL
LIN {X 0,Y 462.543,Z 429.68,A -85,B 0,C 180,E1 -8056.863,E2 -8056.863} C_VEL
LIN {X 0,Y 461.993,Z 424.898,A -85,B 0,C 180,E1 -8059.146,E2 -8059.146} C_VEL
LIN {X 0,Y 460.806,Z 418.294,A -85,B 0,C 180,E1 -8062.474,E2 -8062.474} C_VEL
LIN {X 0,Y 460.52,Z 416.747,A -85,B 0,C 180,E1 -8063.338,E2 -8063.338} C_VEL
LIN {X 0,Y 460.531,Z 416.746,A -85,B 0,C 180,E1 -8066.675,E2 -8066.675} C_VEL
LIN {X 0,Y 460.512,Z 416.75,A -85,B 0,C 180,E1 -8069.76,E2 -8069.76} C_VEL
LIN {X 0,Y 460.581,Z 416.737,A -85,B 0,C 180,E1 -8072.757,E2 -8072.757} C_VEL
LIN {X 0,Y 460.545,Z 416.741,A -85,B 0,C 180,E1 -8075.668,E2 -8075.668} C_VEL
LIN {X 0,Y 460.523,Z 416.743,A -85,B 0,C 180,E1 -8078.578,E2 -8078.578} C_VEL
LIN {X 0,Y 460.593,Z 416.735,A -85,B 0,C 180,E1 -8081.311,E2 -8081.311} C_VEL
LIN {X 0,Y 460.606,Z 416.73,A -85,B 0,C 180,E1 -8084.059,E2 -8084.059} C_VEL
LIN {X 0,Y 460.611,Z 416.735,A -85,B 0,C 180,E1 -8087.666,E2 -8087.666} C_VEL
LIN {X 0,Y 460.622,Z 416.725,A -85,B 0,C 180,E1 -8091.224,E2 -8091.224} C_VEL
LIN {X 0,Y 460.71,Z 416.724,A -85,B 0,C 180,E1 -8093.87,E2 -8093.87} C_VEL
LIN {X 0,Y 460.802,Z 416.703,A -85,B 0,C 180,E1 -8097.378,E2 -8097.378} C_VEL
LIN {X 0,Y 460.856,Z 416.708,A -85,B 0,C 180,E1 -8100,E2 -8100} C_VEL
LIN {X 0,Y 460.802,Z 416.705,A -85,B 0,C 180,E1 -8102.623,E2 -8102.623} C_VEL
LIN {X 0,Y 460.712,Z 416.724,A -85,B 0,C 180,E1 -8106.13,E2 -8106.13} C_VEL
LIN {X 0,Y 460.631,Z 416.724,A -85,B 0,C 180,E1 -8108.776,E2 -8108.776} C_VEL
LIN {X 0,Y 460.615,Z 416.732,A -85,B 0,C 180,E1 -8112.445,E2 -8112.445} C_VEL
LIN {X 0,Y 460.602,Z 416.736,A -85,B 0,C 180,E1 -8115.998,E2 -8115.998} C_VEL
LIN {X 0,Y 460.573,Z 416.733,A -85,B 0,C 180,E1 -8118.902,E2 -8118.902} C_VEL
LIN {X 0,Y 460.518,Z 416.746,A -85,B 0,C 180,E1 -8121.486,E2 -8121.486} C_VEL
LIN {X 0,Y 460.533,Z 416.746,A -85,B 0,C 180,E1 -8124.333,E2 -8124.333} C_VEL
LIN {X 0,Y 460.591,Z 416.736,A -85,B 0,C 180,E1 -8127.748,E2 -8127.748} C_VEL
LIN {X 0,Y 460.523,Z 416.746,A -85,B 0,C 180,E1 -8131.283,E2 -8131.283} C_VEL
LIN {X 0,Y 460.533,Z 416.747,A -85,B 0,C 180,E1 -8134.506,E2 -8134.506} C_VEL
LIN {X 0,Y 460.503,Z 416.749,A -85,B 0,C 180,E1 -8137.623,E2 -8137.623} C_VEL
LIN {X 0,Y 460.545,Z 416.744,A -85,B 0,C 180,E1 -8140.27,E2 -8140.27} C_VEL
LIN {X 0,Y 460.511,Z 416.749,A -85,B 0,C 180,E1 -8143.374,E2 -8143.374} C_VEL
LIN {X 0,Y 460.502,Z 416.753,A -85,B 0,C 180,E1 -8146.625,E2 -8146.625} C_VEL
LIN {X 0,Y 460.558,Z 416.803,A -85,B 0,C 180,E1 -8148.514,E2 -8148.514} C_VEL
LIN {X 0,Y 461.946,Z 424.424,A -85,B 0,C 180,E1 -8150.888,E2 -8150.888} C_VEL
LIN {X 0,Y 462.156,Z 429.801,A -85,B 0,C 180,E1 -8152.535,E2 -8152.535} C_VEL
LIN {X 0,Y 461.727,Z 441.917,A -85,B 0,C 180,E1 -8156.25,E2 -8156.25} C_VEL
LIN {X 0,Y 461.547,Z 451.826,A -85,B 0,C 180,E1 -8159.329,E2 -8159.329} C_VEL
LIN {X 0,Y 461.277,Z 461.895,A -85,B 0,C 180,E1 -8162.44,E2 -8162.44} C_VEL
LIN {X 0,Y 460.98,Z 472.629,A -85,B 0,C 180,E1 -8165.692,E2 -8165.692} C_VEL
LIN {X 0,Y 460.761,Z 482.214,A -85,B 0,C 180,E1 -8168.526,E2 -8168.526} C_VEL
LIN {X 0,Y 460.585,Z 491.295,A -85,B 0,C 180,E1 -8171.116,E2 -8171.116} C_VEL
LIN {X 0,Y 463.908,Z 506.835,A -85,B 0,C 180,E1 -8171.596,E2 -8171.596} C_VEL
LIN {X 0,Y 465.153,Z 513.948,A -85,B 0,C 180,E1 -8171.872,E2 -8171.872} C_VEL
LIN {X 0,Y 464.894,Z 520.11,A -85,B 0,C 180,E1 -8172.096,E2 -8172.096} C_VEL
LIN {X 0,Y 464.111,Z 525.723,A -85,B 0,C 180,E1 -8172.305,E2 -8172.305} C_VEL
LIN {X 0,Y 460.998,Z 534.742,A -85,B 0,C 180,E1 -8172.645,E2 -8172.645} C_VEL
LIN {X 0,Y 457.78,Z 543.488,A -85,B 0,C 180,E1 -8173.067,E2 -8173.067} C_VEL
LIN {X 0,Y 456.839,Z 548.668,A -85,B 0,C 180,E1 -8173.402,E2 -8173.402} C_VEL
LIN {X 0,Y 455.976,Z 560.602,A -85,B 0,C 180,E1 -8174.352,E2 -8174.352} C_VEL
LIN {X 0,Y 455.311,Z 572.007,A -85,B 0,C 180,E1 -8175.473,E2 -8175.473} C_VEL
LIN {X 0,Y 454.555,Z 583.042,A -85,B 0,C 180,E1 -8176.793,E2 -8176.793} C_VEL
LIN {X 0,Y 454.025,Z 592.426,A -85,B 0,C 180,E1 -8178.165,E2 -8178.165} C_VEL
LIN {X 0,Y 453.388,Z 601.185,A -85,B 0,C 180,E1 -8179.731,E2 -8179.731} C_VEL
LIN {X 0,Y 453.056,Z 607.37,A -85,B 0,C 180,E1 -8181.076,E2 -8181.076} C_VEL
LIN {X 0,Y 452.714,Z 613.908,A -85,B 0,C 180,E1 -8182.866,E2 -8182.866} C_VEL
LIN {X 0,Y 452.623,Z 618.815,A -85,B 0,C 180,E1 -8184.654,E2 -8184.654} C_VEL
LIN {X 0,Y 452.479,Z 622.236,A -85,B 0,C 180,E1 -8186.438,E2 -8186.438} C_VEL
LIN {X 0,Y 452.432,Z 624.271,A -85,B 0,C 180,E1 -8188.22,E2 -8188.22} C_VEL
LIN {X 0,Y 452.406,Z 624.975,A -85,B 0,C 180,E1 -8190,E2 -8190} C_VEL
LIN {X 0,Y 452.431,Z 624.348,A -85,B 0,C 180,E1 -8191.78,E2 -8191.78} C_VEL
LIN {X 0,Y 452.478,Z 622.377,A -85,B 0,C 180,E1 -8193.562,E2 -8193.562} C_VEL
LIN {X 0,Y 452.623,Z 619.024,A -85,B 0,C 180,E1 -8195.346,E2 -8195.346} C_VEL
LIN {X 0,Y 452.713,Z 614.192,A -85,B 0,C 180,E1 -8197.134,E2 -8197.134} C_VEL
LIN {X 0,Y 453.02,Z 607.729,A -85,B 0,C 180,E1 -8198.925,E2 -8198.925} C_VEL
LIN {X 0,Y 453.39,Z 600.526,A -85,B 0,C 180,E1 -8200.494,E2 -8200.494} C_VEL
LIN {X 0,Y 454.071,Z 591.559,A -85,B 0,C 180,E1 -8202.061,E2 -8202.061} C_VEL
LIN {X 0,Y 454.651,Z 582.178,A -85,B 0,C 180,E1 -8203.407,E2 -8203.407} C_VEL
LIN {X 0,Y 455.322,Z 571.795,A -85,B 0,C 180,E1 -8204.64,E2 -8204.64} C_VEL
LIN {X 0,Y 456.028,Z 560.34,A -85,B 0,C 180,E1 -8205.761,E2 -8205.761} C_VEL
LIN {X 0,Y 456.889,Z 547.653,A -85,B 0,C 180,E1 -8206.763,E2 -8206.763} C_VEL
LIN {X 0,Y 457.585,Z 534.509,A -85,B 0,C 180,E1 -8207.588,E2 -8207.588} C_VEL
LIN {X 0,Y 458.138,Z 521.51,A -85,B 0,C 180,E1 -8208.214,E2 -8208.214} C_VEL
LIN {X 0,Y 458.216,Z 513.675,A -85,B 0,C 180,E1 -8208.514,E2 -8208.514} C_VEL
LIN {X 0,Y 455.392,Z 499.291,A -85,B 0,C 180,E1 -8209.044,E2 -8209.044} C_VEL
LIN {X 0,Y 453.575,Z 491.249,A -85,B 0,C 180,E1 -8209.288,E2 -8209.288} C_VEL
LIN {X 0,Y 453.782,Z 480.821,A -85,B 0,C 180,E1 -8212.299,E2 -8212.299} C_VEL
LIN {X 0,Y 453.99,Z 471.15,A -85,B 0,C 180,E1 -8215.196,E2 -8215.196} C_VEL
LIN {X 0,Y 454.32,Z 461.529,A -85,B 0,C 180,E1 -8218.146,E2 -8218.146} C_VEL
LIN {X 0,Y 454.559,Z 451.787,A -85,B 0,C 180,E1 -8221.195,E2 -8221.195} C_VEL
LIN {X 0,Y 454.8,Z 441.771,A -85,B 0,C 180,E1 -8224.335,E2 -8224.335} C_VEL
LIN {X 0,Y 455.201,Z 431.378,A -85,B 0,C 180,E1 -8227.547,E2 -8227.547} C_VEL
LIN {X 0,Y 454.981,Z 425.759,A -85,B 0,C 180,E1 -8229.295,E2 -8229.295} C_VEL
LIN {X 0,Y 453.507,Z 417.624,A -85,B 0,C 180,E1 -8231.897,E2 -8231.897} C_VEL
LIN {X 0,Y 453.494,Z 417.625,A -85,B 0,C 180,E1 -8235.47,E2 -8235.47} C_VEL
LIN {X 0,Y 453.484,Z 417.627,A -85,B 0,C 180,E1 -8238.21,E2 -8238.21} C_VEL
LIN {X 0,Y 453.496,Z 417.624,A -85,B 0,C 180,E1 -8240.793,E2 -8240.793} C_VEL
LIN {X 0,Y 453.459,Z 417.626,A -85,B 0,C 180,E1 -8243.917,E2 -8243.917} C_VEL
LIN {X 0,Y 453.485,Z 417.623,A -85,B 0,C 180,E1 -8247.151,E2 -8247.151} C_VEL
LIN {X 0,Y 453.516,Z 417.615,A -85,B 0,C 180,E1 -8250.271,E2 -8250.271} C_VEL
LIN {X 0,Y 453.511,Z 417.619,A -85,B 0,C 180,E1 -8253.294,E2 -8253.294} C_VEL
LIN {X 0,Y 453.506,Z 417.62,A -85,B 0,C 180,E1 -8256.239,E2 -8256.239} C_VEL
LIN {X 0,Y 453.53,Z 417.765,A -85,B 0,C 180,E1 -8258.862,E2 -8258.862} C_VEL
LIN {X 0,Y 458.212,Z 432.024,A -85,B 0,C 180,E1 -8259.745,E2 -8259.745} C_VEL
LIN {X 0,Y 459.005,Z 434.619,A -85,B 0,C 180,E1 -8259.919,E2 -8259.919} C_VEL
LIN {X 0,Y 458.351,Z 448.409,A -85,B 0,C 180,E1 -8260.751,E2 -8260.751} C_VEL
LIN {X 0,Y 457.553,Z 461.962,A -85,B 0,C 180,E1 -8261.762,E2 -8261.762} C_VEL
LIN {X 0,Y 456.67,Z 475.492,A -85,B 0,C 180,E1 -8262.998,E2 -8262.998} C_VEL
LIN {X 0,Y 455.835,Z 487.624,A -85,B 0,C 180,E1 -8264.347,E2 -8264.347} C_VEL
LIN {X 0,Y 455.151,Z 497.795,A -85,B 0,C 180,E1 -8265.696,E2 -8265.696} C_VEL
LIN {X 0,Y 454.452,Z 507.123,A -85,B 0,C 180,E1 -8267.168,E2 -8267.168} C_VEL
LIN {X 0,Y 453.946,Z 515.9,A -85,B 0,C 180,E1 -8268.841,E2 -8268.841} C_VEL
LIN {X 0,Y 453.509,Z 523.539,A -85,B 0,C 180,E1 -8270.635,E2 -8270.635} C_VEL
LIN {X 0,Y 453.175,Z 529.596,A -85,B 0,C 180,E1 -8272.425,E2 -8272.425} C_VEL
LIN {X 0,Y 452.964,Z 533.169,A -85,B 0,C 180,E1 -8273.765,E2 -8273.765} C_VEL
LIN {X 0,Y 452.924,Z 536.841,A -85,B 0,C 180,E1 -8275.55,E2 -8275.55} C_VEL
LIN {X 0,Y 452.741,Z 539.315,A -85,B 0,C 180,E1 -8277.331,E2 -8277.331} C_VEL
LIN {X 0,Y 452.608,Z 540.632,A -85,B 0,C 180,E1 -8279.11,E2 -8279.11} C_VEL
LIN {X 0,Y 452.617,Z 540.761,A -85,B 0,C 180,E1 -8280.89,E2 -8280.89} C_VEL
LIN {X 0,Y 452.762,Z 539.72,A -85,B 0,C 180,E1 -8282.669,E2 -8282.669} C_VEL
LIN {X 0,Y 453.007,Z 537.518,A -85,B 0,C 180,E1 -8284.449,E2 -8284.449} C_VEL
LIN {X 0,Y 453.134,Z 534.123,A -85,B 0,C 180,E1 -8286.233,E2 -8286.233} C_VEL
LIN {X 0,Y 453.379,Z 529.411,A -85,B 0,C 180,E1 -8288.02,E2 -8288.02} C_VEL
LIN {X 0,Y 453.674,Z 523.264,A -85,B 0,C 180,E1 -8289.811,E2 -8289.811} C_VEL
LIN {X 0,Y 454.235,Z 515.455,A -85,B 0,C 180,E1 -8291.603,E2 -8291.603} C_VEL
LIN {X 0,Y 454.794,Z 506.85,A -85,B 0,C 180,E1 -8293.207,E2 -8293.207} C_VEL
LIN {X 0,Y 455.438,Z 498.377,A -85,B 0,C 180,E1 -8294.522,E2 -8294.522} C_VEL
LIN {X 0,Y 456.097,Z 488.085,A -85,B 0,C 180,E1 -8295.873,E2 -8295.873} C_VEL
LIN {X 0,Y 456.908,Z 475.978,A -85,B 0,C 180,E1 -8297.193,E2 -8297.193} C_VEL
LIN {X 0,Y 457.751,Z 463.066,A -85,B 0,C 180,E1 -8298.345,E2 -8298.345} C_VEL
LIN {X 0,Y 458.39,Z 450.818,A -85,B 0,C 180,E1 -8299.247,E2 -8299.247} C_VEL
LIN {X 0,Y 459.066,Z 435.978,A -85,B 0,C 180,E1 -8300.122,E2 -8300.122} C_VEL
LIN {X 0,Y 458.684,Z 433.06,A -85,B 0,C 180,E1 -8300.299,E2 -8300.299} C_VEL
LIN {X 0,Y 454.288,Z 420.062,A -85,B 0,C 180,E1 -8301.119,E2 -8301.119} C_VEL
LIN {X 0,Y 453.506,Z 417.621,A -85,B 0,C 180,E1 -8301.268,E2 -8301.268} C_VEL
LIN {X 0,Y 453.502,Z 417.622,A -85,B 0,C 180,E1 -8304.735,E2 -8304.735} C_VEL
LIN {X 0,Y 453.539,Z 417.62,A -85,B 0,C 180,E1 -8307.961,E2 -8307.961} C_VEL
LIN {X 0,Y 453.468,Z 417.627,A -85,B 0,C 180,E1 -8311.525,E2 -8311.525} C_VEL
LIN {X 0,Y 453.488,Z 417.62,A -85,B 0,C 180,E1 -8314.777,E2 -8314.777} C_VEL
LIN {X 0,Y 453.466,Z 417.625,A -85,B 0,C 180,E1 -8318.312,E2 -8318.312} C_VEL
LIN {X 0,Y 453.495,Z 417.621,A -85,B 0,C 180,E1 -8320.609,E2 -8320.609} C_VEL
LIN {X 0,Y 453.573,Z 417.77,A -85,B 0,C 180,E1 -8323.26,E2 -8323.26} C_VEL
LIN {X 0,Y 453.933,Z 421.881,A -85,B 0,C 180,E1 -8325.055,E2 -8325.055} C_VEL
LIN {X 0,Y 453.424,Z 431.679,A -85,B 0,C 180,E1 -8328.796,E2 -8328.796} C_VEL
LIN {X 0,Y 453.522,Z 439.821,A -85,B 0,C 180,E1 -8331.694,E2 -8331.694} C_VEL
LIN {X 0,Y 453.65,Z 449.603,A -85,B 0,C 180,E1 -8335.026,E2 -8335.026} C_VEL
LIN {X 0,Y 453.605,Z 459.928,A -85,B 0,C 180,E1 -8338.446,E2 -8338.446} C_VEL
LIN {X 0,Y 453.602,Z 469.892,A -85,B 0,C 180,E1 -8341.706,E2 -8341.706} C_VEL
LIN {X 0,Y 453.442,Z 479.31,A -85,B 0,C 180,E1 -8344.771,E2 -8344.771} C_VEL
LIN {X 0,Y 453.305,Z 489.688,A -85,B 0,C 180,E1 -8348.155,E2 -8348.155} C_VEL
LIN {X 0,Y 453.16,Z 497.172,A -85,B 0,C 180,E1 -8350.611,E2 -8350.611} C_VEL
LIN {X 0,Y 455.149,Z 510.601,A -85,B 0,C 180,E1 -8351.044,E2 -8351.044} C_VEL
LIN {X 0,Y 458.002,Z 525.329,A -85,B 0,C 180,E1 -8351.686,E2 -8351.686} C_VEL
LIN {X 0,Y 457.43,Z 540.277,A -85,B 0,C 180,E1 -8352.401,E2 -8352.401} C_VEL
LIN {X 0,Y 456.676,Z 553.66,A -85,B 0,C 180,E1 -8353.229,E2 -8353.229} C_VEL
LIN {X 0,Y 455.853,Z 566.631,A -85,B 0,C 180,E1 -8354.233,E2 -8354.233} C_VEL
LIN {X 0,Y 455.104,Z 578.411,A -85,B 0,C 180,E1 -8355.352,E2 -8355.352} C_VEL
LIN {X 0,Y 454.441,Z 589.15,A -85,B 0,C 180,E1 -8356.586,E2 -8356.586} C_VEL
LIN {X 0,Y 453.951,Z 598.895,A -85,B 0,C 180,E1 -8357.936,E2 -8357.936} C_VEL
LIN {X 0,Y 453.334,Z 608.205,A -85,B 0,C 180,E1 -8359.504,E2 -8359.504} C_VEL
LIN {X 0,Y 452.974,Z 615.744,A -85,B 0,C 180,E1 -8361.074,E2 -8361.074} C_VEL
LIN {X 0,Y 452.737,Z 620.978,A -85,B 0,C 180,E1 -8362.418,E2 -8362.418} C_VEL
LIN {X 0,Y 452.603,Z 626.477,A -85,B 0,C 180,E1 -8364.207,E2 -8364.207} C_VEL
LIN {X 0,Y 452.488,Z 629.515,A -85,B 0,C 180,E1 -8365.546,E2 -8365.546} C_VEL
LIN {X 0,Y 452.491,Z 632.313,A -85,B 0,C 180,E1 -8367.329,E2 -8367.329} C_VEL
LIN {X 0,Y 452.43,Z 633.699,A -85,B 0,C 180,E1 -8369.11,E2 -8369.11} C_VEL
LIN {X 0,Y 452.43,Z 633.707,A -85,B 0,C 180,E1 -8370.89,E2 -8370.89} C_VEL
LIN {X 0,Y 452.491,Z 632.352,A -85,B 0,C 180,E1 -8372.671,E2 -8372.671} C_VEL
LIN {X 0,Y 452.483,Z 629.582,A -85,B 0,C 180,E1 -8374.454,E2 -8374.454} C_VEL
LIN {X 0,Y 452.601,Z 626.566,A -85,B 0,C 180,E1 -8375.793,E2 -8375.793} C_VEL
LIN {X 0,Y 452.667,Z 622.671,A -85,B 0,C 180,E1 -8377.135,E2 -8377.135} C_VEL
LIN {X 0,Y 452.887,Z 617.823,A -85,B 0,C 180,E1 -8378.478,E2 -8378.478} C_VEL
LIN {X 0,Y 453.237,Z 610.884,A -85,B 0,C 180,E1 -8380.046,E2 -8380.046} C_VEL
LIN {X 0,Y 453.748,Z 602.245,A -85,B 0,C 180,E1 -8381.616,E2 -8381.616} C_VEL
LIN {X 0,Y 454.216,Z 593.729,A -85,B 0,C 180,E1 -8382.893,E2 -8382.893} C_VEL
LIN {X 0,Y 454.83,Z 584.334,A -85,B 0,C 180,E1 -8384.085,E2 -8384.085} C_VEL
LIN {X 0,Y 455.593,Z 572.61,A -85,B 0,C 180,E1 -8385.318,E2 -8385.318} C_VEL
LIN {X 0,Y 456.519,Z 559.545,A -85,B 0,C 180,E1 -8386.432,E2 -8386.432} C_VEL
LIN {X 0,Y 457.267,Z 546.184,A -85,B 0,C 180,E1 -8387.339,E2 -8387.339} C_VEL
LIN {X 0,Y 457.974,Z 531.773,A -85,B 0,C 180,E1 -8388.096,E2 -8388.096} C_VEL
LIN {X 0,Y 458.051,Z 524.966,A -85,B 0,C 180,E1 -8388.39,E2 -8388.39} C_VEL
LIN {X 0,Y 455.254,Z 510.662,A -85,B 0,C 180,E1 -8388.994,E2 -8388.994} C_VEL
LIN {X 0,Y 453.169,Z 499.784,A -85,B 0,C 180,E1 -8389.347,E2 -8389.347} C_VEL
LIN {X 0,Y 453.39,Z 491.615,A -85,B 0,C 180,E1 -8392.32,E2 -8392.32} C_VEL
LIN {X 0,Y 453.641,Z 482.48,A -85,B 0,C 180,E1 -8395.708,E2 -8395.708} C_VEL
LIN {X 0,Y 453.982,Z 473.3,A -85,B 0,C 180,E1 -8399.186,E2 -8399.186} C_VEL
LIN {X 0,Y 454.255,Z 465.435,A -85,B 0,C 180,E1 -8402.26,E2 -8402.26} C_VEL
LIN {X 0,Y 454.507,Z 457.506,A -85,B 0,C 180,E1 -8405.44,E2 -8405.44} C_VEL
LIN {X 0,Y 454.761,Z 449.504,A -85,B 0,C 180,E1 -8408.748,E2 -8408.748} C_VEL
LIN {X 0,Y 455.066,Z 442.782,A -85,B 0,C 180,E1 -8411.612,E2 -8411.612} C_VEL
LIN {X 0,Y 455.5,Z 434.631,A -85,B 0,C 180,E1 -8415.214,E2 -8415.214} C_VEL
LIN {X 0,Y 455.553,Z 430.201,A -85,B 0,C 180,E1 -8417.25,E2 -8417.25} C_VEL
LIN {X 0,Y 454.883,Z 425.516,A -85,B 0,C 180,E1 -8419.541,E2 -8419.541} C_VEL
LIN {X 0,Y 453.99,Z 420.419,A -85,B 0,C 180,E1 -8422.14,E2 -8422.14} C_VEL
LIN {X 0,Y 453.463,Z 417.627,A -85,B 0,C 180,E1 -8423.7,E2 -8423.7} C_VEL
LIN {X 0,Y 453.492,Z 417.624,A -85,B 0,C 180,E1 -8426.811,E2 -8426.811} C_VEL
LIN {X 0,Y 453.477,Z 417.626,A -85,B 0,C 180,E1 -8430.268,E2 -8430.268} C_VEL
LIN {X 0,Y 453.511,Z 417.612,A -85,B 0,C 180,E1 -8433.294,E2 -8433.294} C_VEL
LIN {X 0,Y 453.506,Z 417.621,A -85,B 0,C 180,E1 -8436.239,E2 -8436.239} C_VEL
LIN {X 0,Y 453.485,Z 417.614,A -85,B 0,C 180,E1 -8439.118,E2 -8439.118} C_VEL
LIN {X 0,Y 453.515,Z 417.621,A -85,B 0,C 180,E1 -8441.945,E2 -8441.945} C_VEL
LIN {X 0,Y 453.542,Z 417.608,A -85,B 0,C 180,E1 -8444.726,E2 -8444.726} C_VEL
LIN {X 0,Y 453.562,Z 417.612,A -85,B 0,C 180,E1 -8448.379,E2 -8448.379} C_VEL
LIN {X 0,Y 453.588,Z 417.601,A -85,B 0,C 180,E1 -8451.087,E2 -8451.087} C_VEL
LIN {X 0,Y 453.676,Z 417.599,A -85,B 0,C 180,E1 -8453.775,E2 -8453.775} C_VEL
LIN {X 0,Y 453.747,Z 417.582,A -85,B 0,C 180,E1 -8457.337,E2 -8457.337} C_VEL
LIN {X 0,Y 453.826,Z 417.583,A -85,B 0,C 180,E1 -8460,E2 -8460} C_VEL
LIN {X 0,Y 453.746,Z 417.583,A -85,B 0,C 180,E1 -8462.663,E2 -8462.663} C_VEL
LIN {X 0,Y 453.68,Z 417.599,A -85,B 0,C 180,E1 -8466.225,E2 -8466.225} C_VEL
LIN {X 0,Y 453.595,Z 417.601,A -85,B 0,C 180,E1 -8468.913,E2 -8468.913} C_VEL
LIN {X 0,Y 453.565,Z 417.609,A -85,B 0,C 180,E1 -8472.529,E2 -8472.529} C_VEL
LIN {X 0,Y 453.547,Z 417.616,A -85,B 0,C 180,E1 -8476.196,E2 -8476.196} C_VEL
LIN {X 0,Y 453.523,Z 417.611,A -85,B 0,C 180,E1 -8479.041,E2 -8479.041} C_VEL
LIN {X 0,Y 453.478,Z 417.622,A -85,B 0,C 180,E1 -8481.836,E2 -8481.836} C_VEL
LIN {X 0,Y 453.503,Z 417.62,A -85,B 0,C 180,E1 -8484.735,E2 -8484.735} C_VEL
LIN {X 0,Y 453.54,Z 417.615,A -85,B 0,C 180,E1 -8487.961,E2 -8487.961} C_VEL
LIN {X 0,Y 453.468,Z 417.627,A -85,B 0,C 180,E1 -8491.525,E2 -8491.525} C_VEL
LIN {X 0,Y 453.489,Z 417.623,A -85,B 0,C 180,E1 -8494.777,E2 -8494.777} C_VEL
LIN {X 0,Y 453.466,Z 417.625,A -85,B 0,C 180,E1 -8498.312,E2 -8498.312} C_VEL
LIN {X 0,Y 453.496,Z 417.625,A -85,B 0,C 180,E1 -8500.609,E2 -8500.609} C_VEL
LIN {X 0,Y 453.465,Z 417.626,A -85,B 0,C 180,E1 -8503.245,E2 -8503.245} C_VEL
LIN {X 0,Y 453.468,Z 417.627,A -85,B 0,C 180,E1 -8505.779,E2 -8505.779} C_VEL
LIN {X 0,Y 453.523,Z 417.814,A -85,B 0,C 180,E1 -8508.291,E2 -8508.291} C_VEL
LIN {X 0,Y 454.93,Z 425.431,A -85,B 0,C 180,E1 -8510.699,E2 -8510.699} C_VEL
LIN {X 0,Y 455.27,Z 429.378,A -85,B 0,C 180,E1 -8511.933,E2 -8511.933} C_VEL
LIN {X 0,Y 454.819,Z 439.736,A -85,B 0,C 180,E1 -8515.129,E2 -8515.129} C_VEL
LIN {X 0,Y 454.607,Z 449.819,A -85,B 0,C 180,E1 -8518.29,E2 -8518.29} C_VEL
LIN {X 0,Y 454.387,Z 459.594,A -85,B 0,C 180,E1 -8521.349,E2 -8521.349} C_VEL
LIN {X 0,Y 454.051,Z 469.235,A -85,B 0,C 180,E1 -8524.317,E2 -8524.317} C_VEL
LIN {X 0,Y 453.857,Z 478.872,A -85,B 0,C 180,E1 -8527.224,E2 -8527.224} C_VEL
LIN {X 0,Y 453.602,Z 490.162,A -85,B 0,C 180,E1 -8530.495,E2 -8530.495} C_VEL
LIN {X 0,Y 453.573,Z 491.291,A -85,B 0,C 180,E1 -8530.814,E2 -8530.814} C_VEL
LIN {X 0,Y 456.965,Z 507.087,A -85,B 0,C 180,E1 -8531.313,E2 -8531.313} C_VEL
LIN {X 0,Y 458.362,Z 514.826,A -85,B 0,C 180,E1 -8531.622,E2 -8531.622} C_VEL
LIN {X 0,Y 457.85,Z 528.16,A -85,B 0,C 180,E1 -8532.175,E2 -8532.175} C_VEL
LIN {X 0,Y 457.274,Z 541.618,A -85,B 0,C 180,E1 -8532.927,E2 -8532.927} C_VEL
LIN {X 0,Y 456.839,Z 548.668,A -85,B 0,C 180,E1 -8533.402,E2 -8533.402} C_VEL
LIN {X 0,Y 455.896,Z 553.795,A -85,B 0,C 180,E1 -8533.761,E2 -8533.761} C_VEL
LIN {X 0,Y 452.612,Z 561.926,A -85,B 0,C 180,E1 -8534.341,E2 -8534.341} C_VEL
LIN {X 0,Y 449.286,Z 569.69,A -85,B 0,C 180,E1 -8534.998,E2 -8534.998} C_VEL
LIN {X 0,Y 448.289,Z 574.148,A -85,B 0,C 180,E1 -8535.474,E2 -8535.474} C_VEL
LIN {X 0,Y 447.431,Z 585.171,A -85,B 0,C 180,E1 -8536.872,E2 -8536.872} C_VEL
LIN {X 0,Y 446.941,Z 593.821,A -85,B 0,C 180,E1 -8538.204,E2 -8538.204} C_VEL
LIN {X 0,Y 446.307,Z 602.34,A -85,B 0,C 180,E1 -8539.796,E2 -8539.796} C_VEL
LIN {X 0,Y 445.908,Z 609.209,A -85,B 0,C 180,E1 -8541.389,E2 -8541.389} C_VEL
LIN {X 0,Y 445.659,Z 613.966,A -85,B 0,C 180,E1 -8542.752,E2 -8542.752} C_VEL
LIN {X 0,Y 445.542,Z 618.874,A -85,B 0,C 180,E1 -8544.569,E2 -8544.569} C_VEL
LIN {X 0,Y 445.379,Z 622.295,A -85,B 0,C 180,E1 -8546.381,E2 -8546.381} C_VEL
LIN {X 0,Y 445.351,Z 624.33,A -85,B 0,C 180,E1 -8548.191,E2 -8548.191} C_VEL
LIN {X 0,Y 445.315,Z 625.033,A -85,B 0,C 180,E1 -8550,E2 -8550} C_VEL
LIN {X 0,Y 445.35,Z 624.406,A -85,B 0,C 180,E1 -8551.809,E2 -8551.809} C_VEL
LIN {X 0,Y 445.378,Z 622.435,A -85,B 0,C 180,E1 -8553.619,E2 -8553.619} C_VEL
LIN {X 0,Y 445.542,Z 619.081,A -85,B 0,C 180,E1 -8555.431,E2 -8555.431} C_VEL
LIN {X 0,Y 445.659,Z 614.247,A -85,B 0,C 180,E1 -8557.248,E2 -8557.248} C_VEL
LIN {X 0,Y 445.975,Z 607.783,A -85,B 0,C 180,E1 -8559.067,E2 -8559.067} C_VEL
LIN {X 0,Y 446.373,Z 600.579,A -85,B 0,C 180,E1 -8560.661,E2 -8560.661} C_VEL
LIN {X 0,Y 447.098,Z 591.609,A -85,B 0,C 180,E1 -8562.252,E2 -8562.252} C_VEL
LIN {X 0,Y 447.695,Z 582.226,A -85,B 0,C 180,E1 -8563.62,E2 -8563.62} C_VEL
LIN {X 0,Y 448.416,Z 571.84,A -85,B 0,C 180,E1 -8564.871,E2 -8564.871} C_VEL
LIN {X 0,Y 449.169,Z 560.381,A -85,B 0,C 180,E1 -8566.008,E2 -8566.008} C_VEL
LIN {X 0,Y 450.086,Z 547.687,A -85,B 0,C 180,E1 -8567.024,E2 -8567.024} C_VEL
LIN {X 0,Y 450.779,Z 535.216,A -85,B 0,C 180,E1 -8567.821,E2 -8567.821} C_VEL
LIN {X 0,Y 451.377,Z 521.967,A -85,B 0,C 180,E1 -8568.477,E2 -8568.477} C_VEL
LIN {X 0,Y 451.473,Z 514.832,A -85,B 0,C 180,E1 -8568.761,E2 -8568.761} C_VEL
LIN {X 0,Y 448.603,Z 500.118,A -85,B 0,C 180,E1 -8569.324,E2 -8569.324} C_VEL
LIN {X 0,Y 446.583,Z 491.163,A -85,B 0,C 180,E1 -8569.623,E2 -8569.623} C_VEL
LIN {X 0,Y 446.799,Z 480.718,A -85,B 0,C 180,E1 -8572.667,E2 -8572.667} C_VEL
LIN {X 0,Y 447.098,Z 469.34,A -85,B 0,C 180,E1 -8576.113,E2 -8576.113} C_VEL
LIN {X 0,Y 447.405,Z 459.615,A -85,B 0,C 180,E1 -8579.141,E2 -8579.141} C_VEL
LIN {X 0,Y 447.688,Z 449.739,A -85,B 0,C 180,E1 -8582.259,E2 -8582.259} C_VEL
LIN {X 0,Y 448.018,Z 437.795,A -85,B 0,C 180,E1 -8586.033,E2 -8586.033} C_VEL
LIN {X 0,Y 448.315,Z 430.24,A -85,B 0,C 180,E1 -8588.388,E2 -8588.388} C_VEL
LIN {X 0,Y 447.666,Z 424.983,A -85,B 0,C 180,E1 -8590.066,E2 -8590.066} C_VEL
LIN {X 0,Y 446.441,Z 418.504,A -85,B 0,C 180,E1 -8592.144,E2 -8592.144} C_VEL
LIN {X 0,Y 446.458,Z 418.5,A -85,B 0,C 180,E1 -8595.103,E2 -8595.103} C_VEL
LIN {X 0,Y 446.431,Z 418.506,A -85,B 0,C 180,E1 -8598.609,E2 -8598.609} C_VEL
LIN {X 0,Y 446.447,Z 418.502,A -85,B 0,C 180,E1 -8600.973,E2 -8600.973} C_VEL
LIN {X 0,Y 446.423,Z 418.505,A -85,B 0,C 180,E1 -8604.374,E2 -8604.374} C_VEL
LIN {X 0,Y 446.425,Z 418.504,A -85,B 0,C 180,E1 -8607.638,E2 -8607.638} C_VEL
LIN {X 0,Y 446.471,Z 418.496,A -85,B 0,C 180,E1 -8610.792,E2 -8610.792} C_VEL
LIN {X 0,Y 446.48,Z 418.497,A -85,B 0,C 180,E1 -8613.848,E2 -8613.848} C_VEL
LIN {X 0,Y 446.432,Z 418.5,A -85,B 0,C 180,E1 -8616.823,E2 -8616.823} C_VEL
LIN {X 0,Y 446.45,Z 418.501,A -85,B 0,C 180,E1 -8618.565,E2 -8618.565} C_VEL
LIN {X 0,Y 451.322,Z 433.249,A -85,B 0,C 180,E1 -8619.5,E2 -8619.5} C_VEL
LIN {X 0,Y 452.258,Z 436.595,A -85,B 0,C 180,E1 -8619.725,E2 -8619.725} C_VEL
LIN {X 0,Y 451.539,Z 450.147,A -85,B 0,C 180,E1 -8620.568,E2 -8620.568} C_VEL
LIN {X 0,Y 450.721,Z 463.514,A -85,B 0,C 180,E1 -8621.594,E2 -8621.594} C_VEL
LIN {X 0,Y 449.771,Z 476.867,A -85,B 0,C 180,E1 -8622.846,E2 -8622.846} C_VEL
LIN {X 0,Y 449.002,Z 488.004,A -85,B 0,C 180,E1 -8624.102,E2 -8624.102} C_VEL
LIN {X 0,Y 448.283,Z 498.227,A -85,B 0,C 180,E1 -8625.473,E2 -8625.473} C_VEL
LIN {X 0,Y 447.505,Z 507.942,A -85,B 0,C 180,E1 -8627.023,E2 -8627.023} C_VEL
LIN {X 0,Y 446.992,Z 516.446,A -85,B 0,C 180,E1 -8628.665,E2 -8628.665} C_VEL
LIN {X 0,Y 446.509,Z 524.145,A -85,B 0,C 180,E1 -8630.487,E2 -8630.487} C_VEL
LIN {X 0,Y 446.151,Z 530.245,A -85,B 0,C 180,E1 -8632.305,E2 -8632.305} C_VEL
LIN {X 0,Y 445.941,Z 534.928,A -85,B 0,C 180,E1 -8634.12,E2 -8634.12} C_VEL
LIN {X 0,Y 445.876,Z 537.551,A -85,B 0,C 180,E1 -8635.48,E2 -8635.48} C_VEL
LIN {X 0,Y 445.692,Z 540.051,A -85,B 0,C 180,E1 -8637.288,E2 -8637.288} C_VEL
LIN {X 0,Y 445.55,Z 541.39,A -85,B 0,C 180,E1 -8639.096,E2 -8639.096} C_VEL
LIN {X 0,Y 445.56,Z 541.536,A -85,B 0,C 180,E1 -8640.904,E2 -8640.904} C_VEL
LIN {X 0,Y 445.712,Z 540.508,A -85,B 0,C 180,E1 -8642.711,E2 -8642.711} C_VEL
LIN {X 0,Y 445.985,Z 538.316,A -85,B 0,C 180,E1 -8644.519,E2 -8644.519} C_VEL
LIN {X 0,Y 446.122,Z 534.934,A -85,B 0,C 180,E1 -8646.331,E2 -8646.331} C_VEL
LIN {X 0,Y 446.405,Z 530.229,A -85,B 0,C 180,E1 -8648.146,E2 -8648.146} C_VEL
LIN {X 0,Y 446.714,Z 524.074,A -85,B 0,C 180,E1 -8649.966,E2 -8649.966} C_VEL
LIN {X 0,Y 447.316,Z 516.244,A -85,B 0,C 180,E1 -8651.786,E2 -8651.786} C_VEL
LIN {X 0,Y 447.907,Z 507.784,A -85,B 0,C 180,E1 -8653.387,E2 -8653.387} C_VEL
LIN {X 0,Y 448.72,Z 497.574,A -85,B 0,C 180,E1 -8654.977,E2 -8654.977} C_VEL
LIN {X 0,Y 449.447,Z 486.963,A -85,B 0,C 180,E1 -8656.348,E2 -8656.348} C_VEL
LIN {X 0,Y 450.151,Z 476.858,A -85,B 0,C 180,E1 -8657.444,E2 -8657.444} C_VEL
LIN {X 0,Y 451.057,Z 463.747,A -85,B 0,C 180,E1 -8658.627,E2 -8658.627} C_VEL
LIN {X 0,Y 451.736,Z 451.508,A -85,B 0,C 180,E1 -8659.542,E2 -8659.542} C_VEL
LIN {X 0,Y 452.437,Z 437.304,A -85,B 0,C 180,E1 -8660.396,E2 -8660.396} C_VEL
LIN {X 0,Y 452.149,Z 435.213,A -85,B 0,C 180,E1 -8660.528,E2 -8660.528} C_VEL
LIN {X 0,Y 448.271,Z 423.53,A -85,B 0,C 180,E1 -8661.296,E2 -8661.296} C_VEL
LIN {X 0,Y 446.462,Z 418.5,A -85,B 0,C 180,E1 -8661.618,E2 -8661.618} C_VEL
LIN {X 0,Y 446.445,Z 418.501,A -85,B 0,C 180,E1 -8665.153,E2 -8665.153} C_VEL
LIN {X 0,Y 446.486,Z 418.499,A -85,B 0,C 180,E1 -8668.179,E2 -8668.179} C_VEL
LIN {X 0,Y 446.422,Z 418.504,A -85,B 0,C 180,E1 -8671.775,E2 -8671.775} C_VEL
LIN {X 0,Y 446.43,Z 418.5,A -85,B 0,C 180,E1 -8674.523,E2 -8674.523} C_VEL
LIN {X 0,Y 446.417,Z 418.505,A -85,B 0,C 180,E1 -8678.079,E2 -8678.079} C_VEL
LIN {X 0,Y 446.429,Z 418.502,A -85,B 0,C 180,E1 -8680.918,E2 -8680.918} C_VEL
LIN {X 0,Y 446.484,Z 418.621,A -85,B 0,C 180,E1 -8683,E2 -8683} C_VEL
LIN {X 0,Y 446.914,Z 421.574,A -85,B 0,C 180,E1 -8684.371,E2 -8684.371} C_VEL
LIN {X 0,Y 446.618,Z 426.415,A -85,B 0,C 180,E1 -8686.374,E2 -8686.374} C_VEL
LIN {X 0,Y 446.426,Z 437.26,A -85,B 0,C 180,E1 -8690.48,E2 -8690.48} C_VEL
LIN {X 0,Y 446.507,Z 445.471,A -85,B 0,C 180,E1 -8693.392,E2 -8693.392} C_VEL
LIN {X 0,Y 446.559,Z 453.168,A -85,B 0,C 180,E1 -8696.034,E2 -8696.034} C_VEL
LIN {X 0,Y 446.504,Z 462.674,A -85,B 0,C 180,E1 -8699.233,E2 -8699.233} C_VEL
LIN {X 0,Y 446.486,Z 470.448,A -85,B 0,C 180,E1 -8701.821,E2 -8701.821} C_VEL
LIN {X 0,Y 446.337,Z 479.558,A -85,B 0,C 180,E1 -8704.84,E2 -8704.84} C_VEL
LIN {X 0,Y 446.202,Z 488.453,A -85,B 0,C 180,E1 -8707.789,E2 -8707.789} C_VEL
LIN {X 0,Y 446.083,Z 495.9,A -85,B 0,C 180,E1 -8710.267,E2 -8710.267} C_VEL
LIN {X 0,Y 448.288,Z 511.254,A -85,B 0,C 180,E1 -8710.778,E2 -8710.778} C_VEL
LIN {X 0,Y 451.086,Z 525.874,A -85,B 0,C 180,E1 -8711.454,E2 -8711.454} C_VEL
LIN {X 0,Y 450.608,Z 539.314,A -85,B 0,C 180,E1 -8712.126,E2 -8712.126} C_VEL
LIN {X 0,Y 449.808,Z 552.672,A -85,B 0,C 180,E1 -8712.965,E2 -8712.965} C_VEL
LIN {X 0,Y 448.96,Z 565.623,A -85,B 0,C 180,E1 -8713.984,E2 -8713.984} C_VEL
LIN {X 0,Y 448.171,Z 577.429,A -85,B 0,C 180,E1 -8715.121,E2 -8715.121} C_VEL
LIN {X 0,Y 447.451,Z 588.201,A -85,B 0,C 180,E1 -8716.373,E2 -8716.373} C_VEL
LIN {X 0,Y 446.923,Z 597.959,A -85,B 0,C 180,E1 -8717.743,E2 -8717.743} C_VEL
LIN {X 0,Y 446.381,Z 606.116,A -85,B 0,C 180,E1 -8719.109,E2 -8719.109} C_VEL
LIN {X 0,Y 446.033,Z 612.909,A -85,B 0,C 180,E1 -8720.477,E2 -8720.477} C_VEL
LIN {X 0,Y 445.755,Z 618.546,A -85,B 0,C 180,E1 -8721.842,E2 -8721.842} C_VEL
LIN {X 0,Y 445.557,Z 624.467,A -85,B 0,C 180,E1 -8723.661,E2 -8723.661} C_VEL
LIN {X 0,Y 445.545,Z 626.826,A -85,B 0,C 180,E1 -8724.569,E2 -8724.569} C_VEL
LIN {X 0,Y 445.459,Z 630.368,A -85,B 0,C 180,E1 -8726.382,E2 -8726.382} C_VEL
LIN {X 0,Y 445.408,Z 632.464,A -85,B 0,C 180,E1 -8728.192,E2 -8728.192} C_VEL
LIN {X 0,Y 445.348,Z 633.189,A -85,B 0,C 180,E1 -8730,E2 -8730} C_VEL
LIN {X 0,Y 445.408,Z 632.494,A -85,B 0,C 180,E1 -8731.808,E2 -8731.808} C_VEL
LIN {X 0,Y 445.42,Z 631.69,A -85,B 0,C 180,E1 -8732.713,E2 -8732.713} C_VEL
LIN {X 0,Y 445.408,Z 628.912,A -85,B 0,C 180,E1 -8734.525,E2 -8734.525} C_VEL
LIN {X 0,Y 445.543,Z 627.029,A -85,B 0,C 180,E1 -8735.431,E2 -8735.431} C_VEL
LIN {X 0,Y 445.594,Z 621.991,A -85,B 0,C 180,E1 -8737.249,E2 -8737.249} C_VEL
LIN {X 0,Y 445.932,Z 615.353,A -85,B 0,C 180,E1 -8739.068,E2 -8739.068} C_VEL
LIN {X 0,Y 446.324,Z 607.887,A -85,B 0,C 180,E1 -8740.662,E2 -8740.662} C_VEL
LIN {X 0,Y 446.836,Z 600.203,A -85,B 0,C 180,E1 -8742.029,E2 -8742.029} C_VEL
LIN {X 0,Y 447.405,Z 590.8,A -85,B 0,C 180,E1 -8743.412,E2 -8743.412} C_VEL
LIN {X 0,Y 448.178,Z 579.72,A -85,B 0,C 180,E1 -8744.763,E2 -8744.763} C_VEL
LIN {X 0,Y 448.93,Z 568.324,A -85,B 0,C 180,E1 -8745.9,E2 -8745.9} C_VEL
LIN {X 0,Y 449.827,Z 555.919,A -85,B 0,C 180,E1 -8746.917,E2 -8746.917} C_VEL
LIN {X 0,Y 450.651,Z 542.252,A -85,B 0,C 180,E1 -8747.813,E2 -8747.813} C_VEL
LIN {X 0,Y 451.375,Z 527.974,A -85,B 0,C 180,E1 -8748.531,E2 -8748.531} C_VEL
LIN {X 0,Y 449.571,Z 516.735,A -85,B 0,C 180,E1 -8749.05,E2 -8749.05} C_VEL
LIN {X 0,Y 446.686,Z 502.475,A -85,B 0,C 180,E1 -8749.585,E2 -8749.585} C_VEL
LIN {X 0,Y 446.098,Z 499.145,A -85,B 0,C 180,E1 -8749.682,E2 -8749.682} C_VEL
LIN {X 0,Y 446.333,Z 491.045,A -85,B 0,C 180,E1 -8752.692,E2 -8752.692} C_VEL
LIN {X 0,Y 446.575,Z 483.242,A -85,B 0,C 180,E1 -8755.644,E2 -8755.644} C_VEL
LIN {X 0,Y 446.915,Z 474.096,A -85,B 0,C 180,E1 -8759.176,E2 -8759.176} C_VEL
LIN {X 0,Y 447.209,Z 466.223,A -85,B 0,C 180,E1 -8762.298,E2 -8762.298} C_VEL
LIN {X 0,Y 447.485,Z 458.286,A -85,B 0,C 180,E1 -8765.528,E2 -8765.528} C_VEL
LIN {X 0,Y 447.765,Z 450.285,A -85,B 0,C 180,E1 -8768.89,E2 -8768.89} C_VEL
LIN {X 0,Y 448.085,Z 443.549,A -85,B 0,C 180,E1 -8771.805,E2 -8771.805} C_VEL
LIN {X 0,Y 448.493,Z 436.047,A -85,B 0,C 180,E1 -8775.157,E2 -8775.157} C_VEL
LIN {X 0,Y 448.563,Z 431.188,A -85,B 0,C 180,E1 -8777.425,E2 -8777.425} C_VEL
LIN {X 0,Y 447.687,Z 425.448,A -85,B 0,C 180,E1 -8780.284,E2 -8780.284} C_VEL
LIN {X 0,Y 446.593,Z 419.555,A -85,B 0,C 180,E1 -8783.378,E2 -8783.378} C_VEL
LIN {X 0,Y 446.422,Z 418.503,A -85,B 0,C 180,E1 -8783.996,E2 -8783.996} C_VEL
LIN {X 0,Y 446.449,Z 418.5,A -85,B 0,C 180,E1 -8786.566,E2 -8786.566} C_VEL
LIN {X 0,Y 446.432,Z 418.505,A -85,B 0,C 180,E1 -8789.979,E2 -8789.979} C_VEL
LIN {X 0,Y 446.48,Z 418.492,A -85,B 0,C 180,E1 -8792.839,E2 -8792.839} C_VEL
LIN {X 0,Y 446.467,Z 418.497,A -85,B 0,C 180,E1 -8795.923,E2 -8795.923} C_VEL
LIN {X 0,Y 446.455,Z 418.492,A -85,B 0,C 180,E1 -8798.773,E2 -8798.773} C_VEL
LIN {X 0,Y 446.46,Z 418.497,A -85,B 0,C 180,E1 -8801.649,E2 -8801.649} C_VEL
LIN {X 0,Y 446.51,Z 418.486,A -85,B 0,C 180,E1 -8804.48,E2 -8804.48} C_VEL
LIN {X 0,Y 446.52,Z 418.491,A -85,B 0,C 180,E1 -8808.193,E2 -8808.193} C_VEL
LIN {X 0,Y 446.535,Z 418.479,A -85,B 0,C 180,E1 -8810.945,E2 -8810.945} C_VEL
LIN {X 0,Y 446.643,Z 418.475,A -85,B 0,C 180,E1 -8813.676,E2 -8813.676} C_VEL
LIN {X 0,Y 446.694,Z 418.459,A -85,B 0,C 180,E1 -8817.295,E2 -8817.295} C_VEL
LIN {X 0,Y 446.796,Z 418.459,A -85,B 0,C 180,E1 -8820,E2 -8820} C_VEL
LIN {X 0,Y 446.693,Z 418.46,A -85,B 0,C 180,E1 -8822.705,E2 -8822.705} C_VEL
LIN {X 0,Y 446.649,Z 418.474,A -85,B 0,C 180,E1 -8826.324,E2 -8826.324} C_VEL
LIN {X 0,Y 446.54,Z 418.48,A -85,B 0,C 180,E1 -8829.055,E2 -8829.055} C_VEL
LIN {X 0,Y 446.523,Z 418.486,A -85,B 0,C 180,E1 -8832.73,E2 -8832.73} C_VEL
LIN {X 0,Y 446.498,Z 418.494,A -85,B 0,C 180,E1 -8836.228,E2 -8836.228} C_VEL
LIN {X 0,Y 446.472,Z 418.491,A -85,B 0,C 180,E1 -8839.303,E2 -8839.303} C_VEL
LIN {X 0,Y 446.42,Z 418.502,A -85,B 0,C 180,E1 -8842.2,E2 -8842.2} C_VEL
LIN {X 0,Y 446.446,Z 418.5,A -85,B 0,C 180,E1 -8845.153,E2 -8845.153} C_VEL
LIN {X 0,Y 446.486,Z 418.494,A -85,B 0,C 180,E1 -8848.179,E2 -8848.179} C_VEL
LIN {X 0,Y 446.421,Z 418.504,A -85,B 0,C 180,E1 -8851.775,E2 -8851.775} C_VEL
LIN {X 0,Y 446.431,Z 418.504,A -85,B 0,C 180,E1 -8854.523,E2 -8854.523} C_VEL
LIN {X 0,Y 446.417,Z 418.504,A -85,B 0,C 180,E1 -8858.079,E2 -8858.079} C_VEL
LIN {X 0,Y 446.43,Z 418.504,A -85,B 0,C 180,E1 -8860.918,E2 -8860.918} C_VEL
LIN {X 0,Y 446.425,Z 418.504,A -85,B 0,C 180,E1 -8863.843,E2 -8863.843} C_VEL
LIN {X 0,Y 446.402,Z 418.509,A -85,B 0,C 180,E1 -8866.403,E2 -8866.403} C_VEL
LIN {X 0,Y 446.477,Z 418.629,A -85,B 0,C 180,E1 -8867.999,E2 -8867.999} C_VEL
LIN {X 0,Y 447.802,Z 425.712,A -85,B 0,C 180,E1 -8870.267,E2 -8870.267} C_VEL
LIN {X 0,Y 448.322,Z 431.046,A -85,B 0,C 180,E1 -8871.964,E2 -8871.964} C_VEL
LIN {X 0,Y 447.864,Z 441.226,A -85,B 0,C 180,E1 -8875.142,E2 -8875.142} C_VEL
LIN {X 0,Y 447.675,Z 450.145,A -85,B 0,C 180,E1 -8877.967,E2 -8877.967} C_VEL
LIN {X 0,Y 447.403,Z 460.671,A -85,B 0,C 180,E1 -8881.29,E2 -8881.29} C_VEL
LIN {X 0,Y 447.022,Z 470.641,A -85,B 0,C 180,E1 -8884.383,E2 -8884.383} C_VEL
LIN {X 0,Y 446.823,Z 480.387,A -85,B 0,C 180,E1 -8887.334,E2 -8887.334} C_VEL
LIN {X 0,Y 446.584,Z 491.323,A -85,B 0,C 180,E1 -8890.504,E2 -8890.504} C_VEL
LIN {X 0,Y 449.916,Z 506.562,A -85,B 0,C 180,E1 -8890.994,E2 -8890.994} C_VEL
LIN {X 0,Y 451.589,Z 516.345,A -85,B 0,C 180,E1 -8891.394,E2 -8891.394} C_VEL
LIN {X 0,Y 450.99,Z 529.701,A -85,B 0,C 180,E1 -8891.975,E2 -8891.975} C_VEL
LIN {X 0,Y 450.362,Z 543.066,A -85,B 0,C 180,E1 -8892.753,E2 -8892.753} C_VEL
LIN {X 0,Y 449.599,Z 555.373,A -85,B 0,C 180,E1 -8893.658,E2 -8893.658} C_VEL
LIN {X 0,Y 448.877,Z 565.493,A -85,B 0,C 180,E1 -8894.564,E2 -8894.564} C_VEL
LIN {X 0,Y 448.289,Z 574.148,A -85,B 0,C 180,E1 -8895.474,E2 -8895.474} C_VEL
LIN {X 0,Y 447.374,Z 577.12,A -85,B 0,C 180,E1 -8895.802,E2 -8895.802} C_VEL
LIN {X 0,Y 441.027,Z 586.152,A -85,B 0,C 180,E1 -8896.807,E2 -8896.807} C_VEL
LIN {X 0,Y 440.254,Z 588.763,A -85,B 0,C 180,E1 -8897.182,E2 -8897.182} C_VEL
LIN {X 0,Y 439.749,Z 596.535,A -85,B 0,C 180,E1 -8898.476,E2 -8898.476} C_VEL
LIN {X 0,Y 439.157,Z 604.535,A -85,B 0,C 180,E1 -8900.094,E2 -8900.094} C_VEL
LIN {X 0,Y 438.753,Z 610.971,A -85,B 0,C 180,E1 -8901.711,E2 -8901.711} C_VEL
LIN {X 0,Y 438.506,Z 616.672,A -85,B 0,C 180,E1 -8903.558,E2 -8903.558} C_VEL
LIN {X 0,Y 438.339,Z 620.822,A -85,B 0,C 180,E1 -8905.402,E2 -8905.402} C_VEL
LIN {X 0,Y 438.328,Z 623.54,A -85,B 0,C 180,E1 -8907.243,E2 -8907.243} C_VEL
LIN {X 0,Y 438.228,Z 624.906,A -85,B 0,C 180,E1 -8909.081,E2 -8909.081} C_VEL
LIN {X 0,Y 438.228,Z 624.945,A -85,B 0,C 180,E1 -8910.919,E2 -8910.919} C_VEL
LIN {X 0,Y 438.328,Z 623.647,A -85,B 0,C 180,E1 -8912.757,E2 -8912.757} C_VEL
LIN {X 0,Y 438.339,Z 620.992,A -85,B 0,C 180,E1 -8914.598,E2 -8914.598} C_VEL
LIN {X 0,Y 438.506,Z 616.914,A -85,B 0,C 180,E1 -8916.442,E2 -8916.442} C_VEL
LIN {X 0,Y 438.74,Z 611.285,A -85,B 0,C 180,E1 -8918.289,E2 -8918.289} C_VEL
LIN {X 0,Y 439.069,Z 605.916,A -85,B 0,C 180,E1 -8919.676,E2 -8919.676} C_VEL
LIN {X 0,Y 439.588,Z 598.232,A -85,B 0,C 180,E1 -8921.294,E2 -8921.294} C_VEL
LIN {X 0,Y 440.2,Z 590.201,A -85,B 0,C 180,E1 -8922.681,E2 -8922.681} C_VEL
LIN {X 0,Y 440.881,Z 580.528,A -85,B 0,C 180,E1 -8924.069,E2 -8924.069} C_VEL
LIN {X 0,Y 441.714,Z 569.792,A -85,B 0,C 180,E1 -8925.338,E2 -8925.338} C_VEL
LIN {X 0,Y 442.571,Z 557.88,A -85,B 0,C 180,E1 -8926.49,E2 -8926.49} C_VEL
LIN {X 0,Y 443.394,Z 546.142,A -85,B 0,C 180,E1 -8927.408,E2 -8927.408} C_VEL
LIN {X 0,Y 444.121,Z 533.304,A -85,B 0,C 180,E1 -8928.21,E2 -8928.21} C_VEL
LIN {X 0,Y 444.757,Z 519.531,A -85,B 0,C 180,E1 -8928.864,E2 -8928.864} C_VEL
LIN {X 0,Y 444.623,Z 515.51,A -85,B 0,C 180,E1 -8929.036,E2 -8929.036} C_VEL
LIN {X 0,Y 441.828,Z 500.888,A -85,B 0,C 180,E1 -8929.614,E2 -8929.614} C_VEL
LIN {X 0,Y 439.582,Z 491.178,A -85,B 0,C 180,E1 -8929.941,E2 -8929.941} C_VEL
LIN {X 0,Y 439.825,Z 480.609,A -85,B 0,C 180,E1 -8933.047,E2 -8933.047} C_VEL
LIN {X 0,Y 440.139,Z 469.018,A -85,B 0,C 180,E1 -8936.595,E2 -8936.595} C_VEL
LIN {X 0,Y 440.467,Z 459.327,A -85,B 0,C 180,E1 -8939.645,E2 -8939.645} C_VEL
LIN {X 0,Y 440.755,Z 449.342,A -85,B 0,C 180,E1 -8942.83,E2 -8942.83} C_VEL
LIN {X 0,Y 441.17,Z 437.306,A -85,B 0,C 180,E1 -8946.666,E2 -8946.666} C_VEL
LIN {X 0,Y 441.318,Z 430.828,A -85,B 0,C 180,E1 -8948.709,E2 -8948.709} C_VEL
LIN {X 0,Y 440.332,Z 424.177,A -85,B 0,C 180,E1 -8950.873,E2 -8950.873} C_VEL
LIN {X 0,Y 439.405,Z 419.379,A -85,B 0,C 180,E1 -8952.462,E2 -8952.462} C_VEL
LIN {X 0,Y 439.408,Z 419.379,A -85,B 0,C 180,E1 -8955.271,E2 -8955.271} C_VEL
LIN {X 0,Y 439.391,Z 419.384,A -85,B 0,C 180,E1 -8958.743,E2 -8958.743} C_VEL
LIN {X 0,Y 439.384,Z 419.383,A -85,B 0,C 180,E1 -8961.606,E2 -8961.606} C_VEL
LIN {X 0,Y 439.403,Z 419.377,A -85,B 0,C 180,E1 -8964.844,E2 -8964.844} C_VEL
LIN {X 0,Y 439.376,Z 419.381,A -85,B 0,C 180,E1 -8968.14,E2 -8968.14} C_VEL
LIN {X 0,Y 439.427,Z 419.375,A -85,B 0,C 180,E1 -8971.327,E2 -8971.327} C_VEL
LIN {X 0,Y 439.407,Z 419.376,A -85,B 0,C 180,E1 -8974.415,E2 -8974.415} C_VEL
LIN {X 0,Y 439.368,Z 419.382,A -85,B 0,C 180,E1 -8977.425,E2 -8977.425} C_VEL
LIN {X 0,Y 439.431,Z 419.554,A -85,B 0,C 180,E1 -8978.284,E2 -8978.284} C_VEL
LIN {X 0,Y 444.134,Z 433.661,A -85,B 0,C 180,E1 -8979.196,E2 -8979.196} C_VEL
LIN {X 0,Y 445.434,Z 438.78,A -85,B 0,C 180,E1 -8979.551,E2 -8979.551} C_VEL
LIN {X 0,Y 444.638,Z 453.224,A -85,B 0,C 180,E1 -8980.494,E2 -8980.494} C_VEL
LIN {X 0,Y 443.754,Z 466.164,A -85,B 0,C 180,E1 -8981.533,E2 -8981.533} C_VEL
LIN {X 0,Y 442.875,Z 478.126,A -85,B 0,C 180,E1 -8982.69,E2 -8982.69} C_VEL
LIN {X 0,Y 441.989,Z 490.086,A -85,B 0,C 180,E1 -8984.08,E2 -8984.08} C_VEL
LIN {X 0,Y 441.256,Z 500.12,A -85,B 0,C 180,E1 -8985.472,E2 -8985.472} C_VEL
LIN {X 0,Y 440.488,Z 509.896,A -85,B 0,C 180,E1 -8987.093,E2 -8987.093} C_VEL
LIN {X 0,Y 439.949,Z 518.012,A -85,B 0,C 180,E1 -8988.715,E2 -8988.715} C_VEL
LIN {X 0,Y 439.508,Z 524.726,A -85,B 0,C 180,E1 -8990.334,E2 -8990.334} C_VEL
LIN {X 0,Y 439.148,Z 530.874,A -85,B 0,C 180,E1 -8992.182,E2 -8992.182} C_VEL
LIN {X 0,Y 438.904,Z 535.597,A -85,B 0,C 180,E1 -8994.026,E2 -8994.026} C_VEL
LIN {X 0,Y 438.831,Z 538.255,A -85,B 0,C 180,E1 -8995.407,E2 -8995.407} C_VEL
LIN {X 0,Y 438.645,Z 540.788,A -85,B 0,C 180,E1 -8997.245,E2 -8997.245} C_VEL
LIN {X 0,Y 438.492,Z 542.153,A -85,B 0,C 180,E1 -8999.082,E2 -8999.082} C_VEL
LIN {X 0,Y 438.505,Z 542.32,A -85,B 0,C 180,E1 -9000.918,E2 -9000.918} C_VEL
LIN {X 0,Y 438.665,Z 541.313,A -85,B 0,C 180,E1 -9002.755,E2 -9002.755} C_VEL
LIN {X 0,Y 438.965,Z 539.132,A -85,B 0,C 180,E1 -9004.591,E2 -9004.591} C_VEL
LIN {X 0,Y 439.111,Z 535.757,A -85,B 0,C 180,E1 -9006.433,E2 -9006.433} C_VEL
LIN {X 0,Y 439.436,Z 531.048,A -85,B 0,C 180,E1 -9008.276,E2 -9008.276} C_VEL
LIN {X 0,Y 439.762,Z 524.898,A -85,B 0,C 180,E1 -9010.125,E2 -9010.125} C_VEL
LIN {X 0,Y 440.407,Z 517.09,A -85,B 0,C 180,E1 -9011.973,E2 -9011.973} C_VEL
LIN {X 0,Y 441.053,Z 508.694,A -85,B 0,C 180,E1 -9013.588,E2 -9013.588} C_VEL
LIN {X 0,Y 441.782,Z 499.985,A -85,B 0,C 180,E1 -9014.982,E2 -9014.982} C_VEL
LIN {X 0,Y 442.52,Z 489.665,A -85,B 0,C 180,E1 -9016.374,E2 -9016.374} C_VEL
LIN {X 0,Y 443.424,Z 477.793,A -85,B 0,C 180,E1 -9017.706,E2 -9017.706} C_VEL
LIN {X 0,Y 444.377,Z 464.608,A -85,B 0,C 180,E1 -9018.918,E2 -9018.918} C_VEL
LIN {X 0,Y 445.109,Z 452.323,A -85,B 0,C 180,E1 -9019.845,E2 -9019.845} C_VEL
LIN {X 0,Y 445.799,Z 438.652,A -85,B 0,C 180,E1 -9020.681,E2 -9020.681} C_VEL
LIN {X 0,Y 443.305,Z 430.02,A -85,B 0,C 180,E1 -9021.287,E2 -9021.287} C_VEL
LIN {X 0,Y 439.393,Z 419.381,A -85,B 0,C 180,E1 -9022.006,E2 -9022.006} C_VEL
LIN {X 0,Y 439.411,Z 419.378,A -85,B 0,C 180,E1 -9024.573,E2 -9024.573} C_VEL
LIN {X 0,Y 439.443,Z 419.377,A -85,B 0,C 180,E1 -9027.632,E2 -9027.632} C_VEL
LIN {X 0,Y 439.363,Z 419.38,A -85,B 0,C 180,E1 -9030.788,E2 -9030.788} C_VEL
LIN {X 0,Y 439.388,Z 419.38,A -85,B 0,C 180,E1 -9034.044,E2 -9034.044} C_VEL
LIN {X 0,Y 439.349,Z 419.383,A -85,B 0,C 180,E1 -9036.887,E2 -9036.887} C_VEL
LIN {X 0,Y 439.414,Z 419.377,A -85,B 0,C 180,E1 -9039.851,E2 -9039.851} C_VEL
LIN {X 0,Y 439.45,Z 419.571,A -85,B 0,C 180,E1 -9042.775,E2 -9042.775} C_VEL
LIN {X 0,Y 439.94,Z 423.544,A -85,B 0,C 180,E1 -9044.66,E2 -9044.66} C_VEL
LIN {X 0,Y 439.411,Z 431.165,A -85,B 0,C 180,E1 -9047.797,E2 -9047.797} C_VEL
LIN {X 0,Y 439.402,Z 439.091,A -85,B 0,C 180,E1 -9050.818,E2 -9050.818} C_VEL
LIN {X 0,Y 439.463,Z 447.122,A -85,B 0,C 180,E1 -9053.721,E2 -9053.721} C_VEL
LIN {X 0,Y 439.462,Z 455.536,A -85,B 0,C 180,E1 -9056.662,E2 -9056.662} C_VEL
LIN {X 0,Y 439.393,Z 464.517,A -85,B 0,C 180,E1 -9059.737,E2 -9059.737} C_VEL
LIN {X 0,Y 439.376,Z 471.14,A -85,B 0,C 180,E1 -9061.981,E2 -9061.981} C_VEL
LIN {X 0,Y 439.257,Z 479.827,A -85,B 0,C 180,E1 -9064.913,E2 -9064.913} C_VEL
LIN {X 0,Y 439.121,Z 490.164,A -85,B 0,C 180,E1 -9068.401,E2 -9068.401} C_VEL
LIN {X 0,Y 439.016,Z 494.55,A -85,B 0,C 180,E1 -9069.885,E2 -9069.885} C_VEL
LIN {X 0,Y 441.419,Z 511.821,A -85,B 0,C 180,E1 -9070.504,E2 -9070.504} C_VEL
LIN {X 0,Y 444.33,Z 527.716,A -85,B 0,C 180,E1 -9071.29,E2 -9071.29} C_VEL
LIN {X 0,Y 443.599,Z 541.613,A -85,B 0,C 180,E1 -9072.032,E2 -9072.032} C_VEL
LIN {X 0,Y 442.576,Z 558.151,A -85,B 0,C 180,E1 -9073.154,E2 -9073.154} C_VEL
LIN {X 0,Y 441.718,Z 570.439,A -85,B 0,C 180,E1 -9074.189,E2 -9074.189} C_VEL
LIN {X 0,Y 441.054,Z 580.523,A -85,B 0,C 180,E1 -9075.229,E2 -9075.229} C_VEL
LIN {X 0,Y 440.39,Z 590.087,A -85,B 0,C 180,E1 -9076.409,E2 -9076.409} C_VEL
LIN {X 0,Y 439.849,Z 599.324,A -85,B 0,C 180,E1 -9077.777,E2 -9077.777} C_VEL
LIN {X 0,Y 439.278,Z 607.108,A -85,B 0,C 180,E1 -9079.165,E2 -9079.165} C_VEL
LIN {X 0,Y 438.863,Z 614.54,A -85,B 0,C 180,E1 -9080.785,E2 -9080.785} C_VEL
LIN {X 0,Y 438.599,Z 619.693,A -85,B 0,C 180,E1 -9082.172,E2 -9082.172} C_VEL
LIN {X 0,Y 438.448,Z 624.802,A -85,B 0,C 180,E1 -9083.909,E2 -9083.909} C_VEL
LIN {X 0,Y 438.346,Z 628.065,A -85,B 0,C 180,E1 -9085.402,E2 -9085.402} C_VEL
LIN {X 0,Y 438.364,Z 630.863,A -85,B 0,C 180,E1 -9087.243,E2 -9087.243} C_VEL
LIN {X 0,Y 438.313,Z 632.298,A -85,B 0,C 180,E1 -9089.081,E2 -9089.081} C_VEL
LIN {X 0,Y 438.289,Z 632.5,A -85,B 0,C 180,E1 -9090,E2 -9090} C_VEL
LIN {X 0,Y 438.357,Z 631.806,A -85,B 0,C 180,E1 -9091.838,E2 -9091.838} C_VEL
LIN {X 0,Y 438.351,Z 631.026,A -85,B 0,C 180,E1 -9092.757,E2 -9092.757} C_VEL
LIN {X 0,Y 438.336,Z 628.228,A -85,B 0,C 180,E1 -9094.598,E2 -9094.598} C_VEL
LIN {X 0,Y 438.423,Z 625.01,A -85,B 0,C 180,E1 -9096.058,E2 -9096.058} C_VEL
LIN {X 0,Y 438.521,Z 621.31,A -85,B 0,C 180,E1 -9097.366,E2 -9097.366} C_VEL
LIN {X 0,Y 438.859,Z 614.7,A -85,B 0,C 180,E1 -9099.215,E2 -9099.215} C_VEL
LIN {X 0,Y 439.285,Z 607.222,A -85,B 0,C 180,E1 -9100.835,E2 -9100.835} C_VEL
LIN {X 0,Y 439.928,Z 598.087,A -85,B 0,C 180,E1 -9102.455,E2 -9102.455} C_VEL
LIN {X 0,Y 440.408,Z 590.422,A -85,B 0,C 180,E1 -9103.591,E2 -9103.591} C_VEL
LIN {X 0,Y 441.187,Z 579.073,A -85,B 0,C 180,E1 -9105.002,E2 -9105.002} C_VEL
LIN {X 0,Y 442.069,Z 567.735,A -85,B 0,C 180,E1 -9106.154,E2 -9106.154} C_VEL
LIN {X 0,Y 442.974,Z 555.353,A -85,B 0,C 180,E1 -9107.187,E2 -9107.187} C_VEL
LIN {X 0,Y 443.83,Z 541.748,A -85,B 0,C 180,E1 -9108.096,E2 -9108.096} C_VEL
LIN {X 0,Y 444.58,Z 528.496,A -85,B 0,C 180,E1 -9108.782,E2 -9108.782} C_VEL
LIN {X 0,Y 442.201,Z 514.963,A -85,B 0,C 180,E1 -9109.436,E2 -9109.436} C_VEL
LIN {X 0,Y 439.1,Z 499.494,A -85,B 0,C 180,E1 -9110.012,E2 -9110.012} C_VEL
LIN {X 0,Y 439.013,Z 498.479,A -85,B 0,C 180,E1 -9110.04,E2 -9110.04} C_VEL
LIN {X 0,Y 439.27,Z 490.482,A -85,B 0,C 180,E1 -9113.078,E2 -9113.078} C_VEL
LIN {X 0,Y 439.512,Z 482.893,A -85,B 0,C 180,E1 -9116.009,E2 -9116.009} C_VEL
LIN {X 0,Y 439.856,Z 474.87,A -85,B 0,C 180,E1 -9119.165,E2 -9119.165} C_VEL
LIN {X 0,Y 440.158,Z 467.344,A -85,B 0,C 180,E1 -9122.194,E2 -9122.194} C_VEL
LIN {X 0,Y 440.394,Z 460.38,A -85,B 0,C 180,E1 -9125.065,E2 -9125.065} C_VEL
LIN {X 0,Y 440.639,Z 453.711,A -85,B 0,C 180,E1 -9127.884,E2 -9127.884} C_VEL
LIN {X 0,Y 440.994,Z 446.988,A -85,B 0,C 180,E1 -9130.799,E2 -9130.799} C_VEL
LIN {X 0,Y 441.286,Z 440.455,A -85,B 0,C 180,E1 -9133.724,E2 -9133.724} C_VEL
LIN {X 0,Y 441.651,Z 434.886,A -85,B 0,C 180,E1 -9136.29,E2 -9136.29} C_VEL
LIN {X 0,Y 441.338,Z 430.439,A -85,B 0,C 180,E1 -9138.456,E2 -9138.456} C_VEL
LIN {X 0,Y 440.303,Z 424.524,A -85,B 0,C 180,E1 -9141.501,E2 -9141.501} C_VEL
LIN {X 0,Y 439.398,Z 419.377,A -85,B 0,C 180,E1 -9144.359,E2 -9144.359} C_VEL
LIN {X 0,Y 439.374,Z 419.382,A -85,B 0,C 180,E1 -9147.054,E2 -9147.054} C_VEL
LIN {X 0,Y 439.384,Z 419.381,A -85,B 0,C 180,E1 -9150.274,E2 -9150.274} C_VEL
LIN {X 0,Y 439.431,Z 419.364,A -85,B 0,C 180,E1 -9153.396,E2 -9153.396} C_VEL
LIN {X 0,Y 439.389,Z 419.378,A -85,B 0,C 180,E1 -9156.43,E2 -9156.43} C_VEL
LIN {X 0,Y 439.391,Z 419.368,A -85,B 0,C 180,E1 -9159.397,E2 -9159.397} C_VEL
LIN {X 0,Y 439.434,Z 419.373,A -85,B 0,C 180,E1 -9162.31,E2 -9162.31} C_VEL
LIN {X 0,Y 439.449,Z 419.361,A -85,B 0,C 180,E1 -9165.174,E2 -9165.174} C_VEL
LIN {X 0,Y 439.486,Z 419.369,A -85,B 0,C 180,E1 -9168.001,E2 -9168.001} C_VEL
LIN {X 0,Y 439.498,Z 419.355,A -85,B 0,C 180,E1 -9170.798,E2 -9170.798} C_VEL
LIN {X 0,Y 439.615,Z 419.349,A -85,B 0,C 180,E1 -9173.575,E2 -9173.575} C_VEL
LIN {X 0,Y 439.643,Z 419.337,A -85,B 0,C 180,E1 -9177.251,E2 -9177.251} C_VEL
LIN {X 0,Y 439.766,Z 419.334,A -85,B 0,C 180,E1 -9180,E2 -9180} C_VEL
LIN {X 0,Y 439.642,Z 419.338,A -85,B 0,C 180,E1 -9182.749,E2 -9182.749} C_VEL
LIN {X 0,Y 439.62,Z 419.348,A -85,B 0,C 180,E1 -9186.425,E2 -9186.425} C_VEL
LIN {X 0,Y 439.502,Z 419.358,A -85,B 0,C 180,E1 -9189.202,E2 -9189.202} C_VEL
LIN {X 0,Y 439.468,Z 419.365,A -85,B 0,C 180,E1 -9192.938,E2 -9192.938} C_VEL
LIN {X 0,Y 439.45,Z 419.373,A -85,B 0,C 180,E1 -9196.349,E2 -9196.349} C_VEL
LIN {X 0,Y 439.405,Z 419.375,A -85,B 0,C 180,E1 -9199.626,E2 -9199.626} C_VEL
LIN {X 0,Y 439.366,Z 419.377,A -85,B 0,C 180,E1 -9202.576,E2 -9202.576} C_VEL
LIN {X 0,Y 439.4,Z 419.377,A -85,B 0,C 180,E1 -9205.585,E2 -9205.585} C_VEL
LIN {X 0,Y 439.419,Z 419.376,A -85,B 0,C 180,E1 -9208.673,E2 -9208.673} C_VEL
LIN {X 0,Y 439.372,Z 419.38,A -85,B 0,C 180,E1 -9212.031,E2 -9212.031} C_VEL
LIN {X 0,Y 439.396,Z 419.375,A -85,B 0,C 180,E1 -9215.34,E2 -9215.34} C_VEL
LIN {X 0,Y 439.385,Z 419.379,A -85,B 0,C 180,E1 -9218.595,E2 -9218.595} C_VEL
LIN {X 0,Y 439.391,Z 419.379,A -85,B 0,C 180,E1 -9221.257,E2 -9221.257} C_VEL
LIN {X 0,Y 439.407,Z 419.377,A -85,B 0,C 180,E1 -9224.729,E2 -9224.729} C_VEL
LIN {X 0,Y 439.438,Z 419.528,A -85,B 0,C 180,E1 -9227.716,E2 -9227.716} C_VEL
LIN {X 0,Y 440.977,Z 427.758,A -85,B 0,C 180,E1 -9230.395,E2 -9230.395} C_VEL
LIN {X 0,Y 441.385,Z 431.508,A -85,B 0,C 180,E1 -9231.612,E2 -9231.612} C_VEL
LIN {X 0,Y 440.964,Z 440.293,A -85,B 0,C 180,E1 -9234.373,E2 -9234.373} C_VEL
LIN {X 0,Y 440.714,Z 450.666,A -85,B 0,C 180,E1 -9237.692,E2 -9237.692} C_VEL
LIN {X 0,Y 440.428,Z 460.657,A -85,B 0,C 180,E1 -9240.877,E2 -9240.877} C_VEL
LIN {X 0,Y 440.079,Z 470.453,A -85,B 0,C 180,E1 -9243.949,E2 -9243.949} C_VEL
LIN {X 0,Y 439.84,Z 480.28,A -85,B 0,C 180,E1 -9246.954,E2 -9246.954} C_VEL
LIN {X 0,Y 439.577,Z 491.289,A -85,B 0,C 180,E1 -9250.181,E2 -9250.181} C_VEL
LIN {X 0,Y 442.888,Z 506.229,A -85,B 0,C 180,E1 -9250.67,E2 -9250.67} C_VEL
LIN {X 0,Y 444.843,Z 517.146,A -85,B 0,C 180,E1 -9251.133,E2 -9251.133} C_VEL
LIN {X 0,Y 444.215,Z 530.306,A -85,B 0,C 180,E1 -9251.722,E2 -9251.722} C_VEL
LIN {X 0,Y 443.585,Z 543.111,A -85,B 0,C 180,E1 -9252.481,E2 -9252.481} C_VEL
LIN {X 0,Y 442.756,Z 555.423,A -85,B 0,C 180,E1 -9253.398,E2 -9253.398} C_VEL
LIN {X 0,Y 441.974,Z 565.546,A -85,B 0,C 180,E1 -9254.316,E2 -9254.316} C_VEL
LIN {X 0,Y 441.223,Z 576.104,A -85,B 0,C 180,E1 -9255.471,E2 -9255.471} C_VEL
LIN {X 0,Y 440.452,Z 585.771,A -85,B 0,C 180,E1 -9256.74,E2 -9256.74} C_VEL
LIN {X 0,Y 440.254,Z 588.763,A -85,B 0,C 180,E1 -9257.182,E2 -9257.182} C_VEL
LIN {X 0,Y 439.454,Z 592.57,A -85,B 0,C 180,E1 -9257.77,E2 -9257.77} C_VEL
LIN {X 0,Y 436.185,Z 598.375,A -85,B 0,C 180,E1 -9258.731,E2 -9258.731} C_VEL
LIN {X 0,Y 432.862,Z 603.711,A -85,B 0,C 180,E1 -9259.747,E2 -9259.747} C_VEL
LIN {X 0,Y 431.988,Z 606.62,A -85,B 0,C 180,E1 -9260.414,E2 -9260.414} C_VEL
LIN {X 0,Y 431.604,Z 612.618,A -85,B 0,C 180,E1 -9262.044,E2 -9262.044} C_VEL
LIN {X 0,Y 431.435,Z 617.001,A -85,B 0,C 180,E1 -9263.556,E2 -9263.556} C_VEL
LIN {X 0,Y 431.269,Z 620.881,A -85,B 0,C 180,E1 -9265.326,E2 -9265.326} C_VEL
LIN {X 0,Y 431.225,Z 623.599,A -85,B 0,C 180,E1 -9267.197,E2 -9267.197} C_VEL
LIN {X 0,Y 431.146,Z 624.964,A -85,B 0,C 180,E1 -9269.066,E2 -9269.066} C_VEL
LIN {X 0,Y 431.146,Z 625.003,A -85,B 0,C 180,E1 -9270.934,E2 -9270.934} C_VEL
LIN {X 0,Y 431.224,Z 623.705,A -85,B 0,C 180,E1 -9272.802,E2 -9272.802} C_VEL
LIN {X 0,Y 431.269,Z 621.049,A -85,B 0,C 180,E1 -9274.674,E2 -9274.674} C_VEL
LIN {X 0,Y 431.439,Z 616.97,A -85,B 0,C 180,E1 -9276.548,E2 -9276.548} C_VEL
LIN {X 0,Y 431.675,Z 611.34,A -85,B 0,C 180,E1 -9278.426,E2 -9278.426} C_VEL
LIN {X 0,Y 432.031,Z 605.97,A -85,B 0,C 180,E1 -9279.835,E2 -9279.835} C_VEL
LIN {X 0,Y 432.621,Z 598.284,A -85,B 0,C 180,E1 -9281.479,E2 -9281.479} C_VEL
LIN {X 0,Y 433.212,Z 590.252,A -85,B 0,C 180,E1 -9282.889,E2 -9282.889} C_VEL
LIN {X 0,Y 433.961,Z 580.576,A -85,B 0,C 180,E1 -9284.299,E2 -9284.299} C_VEL
LIN {X 0,Y 434.828,Z 569.837,A -85,B 0,C 180,E1 -9285.587,E2 -9285.587} C_VEL
LIN {X 0,Y 435.752,Z 557.919,A -85,B 0,C 180,E1 -9286.756,E2 -9286.756} C_VEL
LIN {X 0,Y 436.618,Z 546.174,A -85,B 0,C 180,E1 -9287.687,E2 -9287.687} C_VEL
LIN {X 0,Y 437.378,Z 533.325,A -85,B 0,C 180,E1 -9288.501,E2 -9288.501} C_VEL
LIN {X 0,Y 438.06,Z 519.14,A -85,B 0,C 180,E1 -9289.181,E2 -9289.181} C_VEL
LIN {X 0,Y 436.973,Z 511.549,A -85,B 0,C 180,E1 -9289.524,E2 -9289.524} C_VEL
LIN {X 0,Y 434.085,Z 497.546,A -85,B 0,C 180,E1 -9290.054,E2 -9290.054} C_VEL
LIN {X 0,Y 432.583,Z 491.234,A -85,B 0,C 180,E1 -9290.259,E2 -9290.259} C_VEL
LIN {X 0,Y 432.833,Z 480.502,A -85,B 0,C 180,E1 -9293.441,E2 -9293.441} C_VEL
LIN {X 0,Y 433.188,Z 468.935,A -85,B 0,C 180,E1 -9297.018,E2 -9297.018} C_VEL
LIN {X 0,Y 433.508,Z 459.033,A -85,B 0,C 180,E1 -9300.17,E2 -9300.17} C_VEL
LIN {X 0,Y 433.831,Z 448.934,A -85,B 0,C 180,E1 -9303.422,E2 -9303.422} C_VEL
LIN {X 0,Y 434.35,Z 436.097,A -85,B 0,C 180,E1 -9307.548,E2 -9307.548} C_VEL
LIN {X 0,Y 434.295,Z 431.171,A -85,B 0,C 180,E1 -9309.133,E2 -9309.133} C_VEL
LIN {X 0,Y 432.941,Z 423.31,A -85,B 0,C 180,E1 -9311.725,E2 -9311.725} C_VEL
LIN {X 0,Y 432.33,Z 420.26,A -85,B 0,C 180,E1 -9312.768,E2 -9312.768} C_VEL
LIN {X 0,Y 432.343,Z 420.261,A -85,B 0,C 180,E1 -9315.663,E2 -9315.663} C_VEL
LIN {X 0,Y 432.336,Z 420.261,A -85,B 0,C 180,E1 -9318.398,E2 -9318.398} C_VEL
LIN {X 0,Y 432.347,Z 420.261,A -85,B 0,C 180,E1 -9321.851,E2 -9321.851} C_VEL
LIN {X 0,Y 432.343,Z 420.255,A -85,B 0,C 180,E1 -9325.323,E2 -9325.323} C_VEL
LIN {X 0,Y 432.326,Z 420.258,A -85,B 0,C 180,E1 -9328.654,E2 -9328.654} C_VEL
LIN {X 0,Y 432.383,Z 420.253,A -85,B 0,C 180,E1 -9331.369,E2 -9331.369} C_VEL
LIN {X 0,Y 432.367,Z 420.254,A -85,B 0,C 180,E1 -9333.968,E2 -9333.968} C_VEL
LIN {X 0,Y 432.322,Z 420.258,A -85,B 0,C 180,E1 -9337.036,E2 -9337.036} C_VEL
LIN {X 0,Y 432.348,Z 420.318,A -85,B 0,C 180,E1 -9337.974,E2 -9337.974} C_VEL
LIN {X 0,Y 436.95,Z 434.192,A -85,B 0,C 180,E1 -9338.889,E2 -9338.889} C_VEL
LIN {X 0,Y 438.459,Z 438.841,A -85,B 0,C 180,E1 -9339.23,E2 -9339.23} C_VEL
LIN {X 0,Y 438.343,Z 446.394,A -85,B 0,C 180,E1 -9339.713,E2 -9339.713} C_VEL
LIN {X 0,Y 437.495,Z 459.304,A -85,B 0,C 180,E1 -9340.651,E2 -9340.651} C_VEL
LIN {X 0,Y 436.539,Z 472.107,A -85,B 0,C 180,E1 -9341.78,E2 -9341.78} C_VEL
LIN {X 0,Y 435.581,Z 484.614,A -85,B 0,C 180,E1 -9343.116,E2 -9343.116} C_VEL
LIN {X 0,Y 434.786,Z 495.635,A -85,B 0,C 180,E1 -9344.531,E2 -9344.531} C_VEL
LIN {X 0,Y 433.904,Z 506.085,A -85,B 0,C 180,E1 -9346.137,E2 -9346.137} C_VEL
LIN {X 0,Y 433.353,Z 514.047,A -85,B 0,C 180,E1 -9347.591,E2 -9347.591} C_VEL
LIN {X 0,Y 432.763,Z 521.577,A -85,B 0,C 180,E1 -9349.236,E2 -9349.236} C_VEL
LIN {X 0,Y 432.327,Z 528.568,A -85,B 0,C 180,E1 -9351.116,E2 -9351.116} C_VEL
LIN {X 0,Y 431.987,Z 533.891,A -85,B 0,C 180,E1 -9352.937,E2 -9352.937} C_VEL
LIN {X 0,Y 431.862,Z 537.208,A -85,B 0,C 180,E1 -9354.396,E2 -9354.396} C_VEL
LIN {X 0,Y 431.751,Z 540.377,A -85,B 0,C 180,E1 -9356.267,E2 -9356.267} C_VEL
LIN {X 0,Y 431.484,Z 542.367,A -85,B 0,C 180,E1 -9358.133,E2 -9358.133} C_VEL
LIN {X 0,Y 431.435,Z 543.16,A -85,B 0,C 180,E1 -9360,E2 -9360} C_VEL
LIN {X 0,Y 431.523,Z 542.757,A -85,B 0,C 180,E1 -9361.867,E2 -9361.867} C_VEL
LIN {X 0,Y 431.772,Z 541.184,A -85,B 0,C 180,E1 -9363.733,E2 -9363.733} C_VEL
LIN {X 0,Y 431.965,Z 538.434,A -85,B 0,C 180,E1 -9365.602,E2 -9365.602} C_VEL
LIN {X 0,Y 432.228,Z 534.428,A -85,B 0,C 180,E1 -9367.474,E2 -9367.474} C_VEL
LIN {X 0,Y 432.684,Z 529.026,A -85,B 0,C 180,E1 -9369.348,E2 -9369.348} C_VEL
LIN {X 0,Y 432.942,Z 524.03,A -85,B 0,C 180,E1 -9370.759,E2 -9370.759} C_VEL
LIN {X 0,Y 433.622,Z 516.874,A -85,B 0,C 180,E1 -9372.401,E2 -9372.401} C_VEL
LIN {X 0,Y 434.354,Z 508.205,A -85,B 0,C 180,E1 -9374.046,E2 -9374.046} C_VEL
LIN {X 0,Y 435.093,Z 499.294,A -85,B 0,C 180,E1 -9375.457,E2 -9375.457} C_VEL
LIN {X 0,Y 435.954,Z 488.685,A -85,B 0,C 180,E1 -9376.869,E2 -9376.869} C_VEL
LIN {X 0,Y 436.85,Z 477.1,A -85,B 0,C 180,E1 -9378.15,E2 -9378.15} C_VEL
LIN {X 0,Y 437.813,Z 464.13,A -85,B 0,C 180,E1 -9379.334,E2 -9379.334} C_VEL
LIN {X 0,Y 438.64,Z 451.596,A -85,B 0,C 180,E1 -9380.272,E2 -9380.272} C_VEL
LIN {X 0,Y 439.222,Z 440.143,A -85,B 0,C 180,E1 -9380.98,E2 -9380.98} C_VEL
LIN {X 0,Y 436.01,Z 429.877,A -85,B 0,C 180,E1 -9381.731,E2 -9381.731} C_VEL
LIN {X 0,Y 432.329,Z 420.26,A -85,B 0,C 180,E1 -9382.415,E2 -9382.415} C_VEL
LIN {X 0,Y 432.347,Z 420.258,A -85,B 0,C 180,E1 -9385.001,E2 -9385.001} C_VEL
LIN {X 0,Y 432.384,Z 420.255,A -85,B 0,C 180,E1 -9388.123,E2 -9388.123} C_VEL
LIN {X 0,Y 432.323,Z 420.259,A -85,B 0,C 180,E1 -9391.346,E2 -9391.346} C_VEL
